C03654=1212.601,101.291,-48.958,-178.587,5.743,148.593
C03655=1212.595,101.540,-48.977,-178.585,5.744,148.593
C03656=1212.591,101.790,-48.996,-178.582,5.744,148.592
C03657=1212.586,102.039,-49.014,-178.579,5.746,148.592
C03658=1212.581,102.288,-49.033,-178.577,5.747,148.591
C03659=1212.577,102.537,-49.052,-178.574,5.747,148.591
C03660=1212.571,102.787,-49.070,-178.572,5.748,148.590
C03661=1212.567,103.035,-49.089,-178.569,5.750,148.590
C03662=1212.561,103.286,-49.108,-178.567,5.750,148.589
C03663=1212.557,103.534,-49.127,-178.564,5.751,148.589
C03664=1212.553,103.784,-49.145,-178.561,5.752,148.588
C03665=1212.547,104.033,-49.164,-178.559,5.753,148.588
C03666=1212.543,104.281,-49.183,-178.556,5.754,148.587
C03667=1212.538,104.532,-49.202,-178.553,5.756,148.587
C03668=1212.533,104.780,-49.221,-178.551,5.756,148.586
C03669=1212.528,105.030,-49.240,-178.549,5.757,148.585
C03670=1212.523,105.279,-49.258,-178.545,5.759,148.585
C03671=1212.519,105.529,-49.278,-178.543,5.760,148.584
C03672=1212.514,105.778,-49.296,-178.541,5.760,148.584
C03673=1212.508,106.027,-49.315,-178.537,5.762,148.583
C03674=1212.504,106.276,-49.334,-178.535,5.763,148.583
C03675=1212.499,106.525,-49.353,-178.533,5.763,148.582
C03676=1212.495,106.775,-49.372,-178.530,5.765,148.582
C03677=1212.489,107.043,-49.393,-178.527,5.766,148.581
C03678=1212.484,107.312,-49.413,-178.524,5.767,148.580
C03679=1212.478,107.580,-49.434,-178.522,5.768,148.580
C03680=1212.474,107.849,-49.454,-178.519,5.769,148.579
C03681=1212.469,108.098,-49.473,-178.516,5.770,148.579
C03682=1212.465,108.347,-49.492,-178.514,5.771,148.578
C03683=1212.459,108.596,-49.511,-178.511,5.772,148.578
C03684=1212.454,108.846,-49.530,-178.509,5.773,148.577
C03685=1212.450,109.094,-49.549,-178.506,5.774,148.577
C03686=1212.444,109.343,-49.568,-178.503,5.775,148.576
C03687=1212.440,109.593,-49.587,-178.501,5.776,148.576
C03688=1212.435,109.842,-49.606,-178.498,5.777,148.575
C03689=1212.430,110.092,-49.625,-178.496,5.779,148.575
C03690=1212.426,110.341,-49.645,-178.493,5.779,148.574
C03691=1212.420,110.590,-49.664,-178.491,5.780,148.573
C03692=1212.416,110.839,-49.683,-178.488,5.782,148.573
C03693=1212.411,111.088,-49.702,-178.486,5.783,148.572
C03694=1212.406,111.338,-49.721,-178.483,5.783,148.572
C03695=1212.401,111.587,-49.740,-178.480,5.785,148.571
C03696=1212.397,111.836,-49.759,-178.478,5.786,148.571
C03697=1212.391,112.085,-49.779,-178.475,5.787,148.570
C03698=1212.387,112.334,-49.798,-178.472,5.788,148.570
C03699=1212.382,112.583,-49.817,-178.470,5.789,148.569
C03700=1212.377,112.833,-49.837,-178.467,5.790,148.569
C03701=1212.373,113.081,-49.855,-178.465,5.791,148.568
C03702=1212.368,113.331,-49.875,-178.462,5.792,148.568
C03703=1212.363,113.581,-49.894,-178.459,5.793,148.567
C03704=1212.358,113.830,-49.913,-178.457,5.794,148.567
C03705=1212.354,114.079,-49.932,-178.454,5.796,148.566
C03706=1212.348,114.328,-49.952,-178.452,5.797,148.566
C03707=1212.343,114.578,-49.971,-178.449,5.797,148.565
C03708=1212.339,114.826,-49.990,-178.446,5.799,148.564
C03709=1212.334,115.076,-50.010,-178.444,5.800,148.564
C03710=1212.329,115.325,-50.029,-178.442,5.801,148.563
C03711=1212.324,115.574,-50.049,-178.439,5.802,148.563
C03712=1212.320,115.823,-50.068,-178.436,5.803,148.562
C03713=1212.315,116.072,-50.087,-178.433,5.804,148.562
C03714=1212.310,116.322,-50.107,-178.431,5.805,148.561
C03715=1212.305,116.571,-50.126,-178.429,5.806,148.561
C03716=1212.300,116.820,-50.146,-178.426,5.808,148.560
C03717=1212.296,117.069,-50.165,-178.423,5.808,148.560
C03718=1212.291,117.319,-50.185,-178.421,5.809,148.559
C03719=1212.286,117.567,-50.204,-178.418,5.811,148.559
C03720=1212.281,117.817,-50.224,-178.416,5.812,148.558
C03721=1212.276,118.066,-50.243,-178.413,5.813,148.558
C03722=1212.272,118.315,-50.262,-178.411,5.814,148.557
C03723=1212.267,118.565,-50.282,-178.408,5.815,148.557
C03724=1212.262,118.814,-50.301,-178.405,5.816,148.556
C03725=1212.257,119.062,-50.322,-178.403,5.817,148.556
C03726=1212.253,119.312,-50.341,-178.400,5.819,148.555
C03727=1212.247,119.561,-50.361,-178.397,5.819,148.554
C03728=1212.243,119.810,-50.380,-178.395,5.820,148.554
C03729=1212.239,120.060,-50.399,-178.392,5.822,148.553
C03730=1212.233,120.309,-50.419,-178.390,5.823,148.553
C03731=1212.229,120.558,-50.439,-178.387,5.824,148.553
C03732=1212.224,120.807,-50.459,-178.385,5.825,148.552
C03733=1212.219,121.056,-50.478,-178.382,5.827,148.552
C03734=1212.214,121.306,-50.498,-178.379,5.827,148.551
C03735=1212.209,121.555,-50.517,-178.377,5.828,148.551
C03736=1212.205,121.804,-50.538,-178.374,5.830,148.550
C03737=1212.199,122.053,-50.557,-178.372,5.831,148.550
C03738=1212.195,122.302,-50.576,-178.369,5.832,148.549
C03739=1212.191,122.551,-50.596,-178.367,5.833,148.549
C03740=1212.186,122.800,-50.616,-178.363,5.835,148.548
C03741=1212.181,123.050,-50.635,-178.361,5.836,148.547
C03742=1212.176,123.299,-50.655,-178.359,5.836,148.547
C03743=1212.172,123.548,-50.675,-178.356,5.838,148.546
C03744=1212.166,123.797,-50.695,-178.353,5.839,148.546
C03745=1212.162,124.047,-50.714,-178.351,5.840,148.545
C03746=1212.157,124.295,-50.735,-178.348,5.841,148.545
C03747=1212.152,124.545,-50.754,-178.345,5.843,148.544
C03748=1212.147,124.793,-50.774,-178.343,5.844,148.544
C03749=1212.143,125.043,-50.794,-178.341,5.844,148.543
C03750=1212.138,125.292,-50.814,-178.338,5.846,148.543
C03751=1212.134,125.541,-50.834,-178.335,5.847,148.542
C03752=1212.128,125.790,-50.853,-178.333,5.849,148.542
C03753=1212.124,126.039,-50.874,-178.330,5.849,148.541
C03754=1212.119,126.289,-50.893,-178.327,5.851,148.541
C03755=1212.114,126.538,-50.913,-178.325,5.852,148.540
C03756=1212.110,126.787,-50.933,-178.322,5.853,148.540
C03757=1212.104,127.036,-50.953,-178.320,5.854,148.539
C03758=1212.100,127.285,-50.973,-178.317,5.855,148.539
C03759=1212.095,127.535,-50.993,-178.315,5.857,148.538
C03760=1212.090,127.784,-51.014,-178.312,5.857,148.538
C03761=1212.085,128.033,-51.033,-178.309,5.859,148.537
C03762=1212.080,128.282,-51.053,-178.307,5.860,148.537
C03763=1212.076,128.531,-51.073,-178.304,5.861,148.536
C03764=1212.071,128.780,-51.093,-178.302,5.862,148.536
C03765=1212.066,129.030,-51.113,-178.299,5.864,148.535
C03766=1212.062,129.279,-51.133,-178.297,5.865,148.535
C03767=1212.057,129.528,-51.153,-178.294,5.866,148.534
C03768=1212.052,129.777,-51.173,-178.291,5.867,148.534
C03769=1212.047,130.026,-51.193,-178.289,5.868,148.533
C03770=1212.042,130.275,-51.214,-178.286,5.870,148.533
C03771=1212.038,130.524,-51.234,-178.284,5.870,148.532
C03772=1212.033,130.774,-51.254,-178.281,5.872,148.532
C03773=1212.029,131.023,-51.274,-178.279,5.873,148.532
C03774=1212.023,131.272,-51.293,-178.276,5.874,148.531
C03775=1212.019,131.521,-51.314,-178.273,5.875,148.530
C03776=1212.014,131.770,-51.335,-178.270,5.877,148.530
C03777=1212.009,132.020,-51.354,-178.268,5.878,148.529
C03778=1212.005,132.268,-51.375,-178.265,5.879,148.529
C03779=1212.000,132.517,-51.395,-178.263,5.880,148.528
C03780=1211.995,132.767,-51.415,-178.260,5.882,148.528
C03781=1211.990,133.035,-51.437,-178.258,5.883,148.527
C03782=1211.984,133.304,-51.459,-178.254,5.884,148.527
C03783=1211.980,133.572,-51.481,-178.252,5.886,148.526
C03784=1211.974,133.841,-51.502,-178.249,5.886,148.526
C03785=1211.970,134.090,-51.523,-178.246,5.888,148.525
C03786=1211.965,134.339,-51.543,-178.244,5.889,148.525
C03787=1211.960,134.588,-51.564,-178.241,5.891,148.524
C03788=1211.955,134.838,-51.584,-178.239,5.892,148.524
C03789=1211.951,135.087,-51.604,-178.236,5.893,148.523
C03790=1211.946,135.336,-51.624,-178.234,5.894,148.523
C03791=1211.941,135.585,-51.645,-178.231,5.895,148.522
C03792=1211.937,135.835,-51.665,-178.229,5.896,148.522
C03793=1211.932,136.084,-51.685,-178.226,5.898,148.522
C03794=1211.927,136.333,-51.706,-178.223,5.900,148.521
C03795=1211.922,136.582,-51.727,-178.221,5.901,148.521
C03796=1211.917,136.830,-51.747,-178.217,5.902,148.520
C03797=1211.912,137.079,-51.768,-178.215,5.903,148.520
C03798=1211.907,137.329,-51.787,-178.213,5.905,148.519
C03799=1211.903,137.578,-51.808,-178.210,5.905,148.519
C03800=1211.898,137.827,-51.829,-178.207,5.907,148.518
C03801=1211.893,138.076,-51.849,-178.205,5.908,148.518
C03802=1211.889,138.325,-51.869,-178.202,5.910,148.517
C03803=1211.884,138.574,-51.890,-178.200,5.911,148.517
C03804=1211.879,138.823,-51.911,-178.197,5.912,148.516
C03805=1211.875,139.072,-51.931,-178.195,5.913,148.516
C03806=1211.870,139.321,-51.952,-178.192,5.915,148.515
C03807=1211.865,139.570,-51.972,-178.189,5.915,148.515
C03808=1211.860,139.820,-51.993,-178.187,5.917,148.514
C03809=1211.855,140.069,-52.013,-178.185,5.918,148.514
C03810=1211.851,140.318,-52.033,-178.181,5.920,148.513
C03811=1211.846,140.567,-52.054,-178.179,5.921,148.513
C03812=1211.841,140.816,-52.075,-178.176,5.922,148.512
C03813=1211.836,141.066,-52.096,-178.174,5.923,148.512
C03814=1211.832,141.315,-52.116,-178.171,5.925,148.512
C03815=1211.827,141.564,-52.137,-178.168,5.926,148.511
C03816=1211.823,141.814,-52.158,-178.166,5.927,148.511
C03817=1211.819,142.062,-52.179,-178.163,5.929,148.510
C03818=1211.813,142.311,-52.200,-178.161,5.930,148.510
C03819=1211.809,142.560,-52.220,-178.158,5.931,148.509
C03820=1211.804,142.809,-52.241,-178.156,5.932,148.509
C03821=1211.799,143.058,-52.262,-178.153,5.934,148.508
C03822=1211.794,143.308,-52.283,-178.151,5.935,148.508
C03823=1211.790,143.556,-52.303,-178.148,5.937,148.507
C03824=1211.785,143.806,-52.324,-178.145,5.937,148.507
C03825=1211.780,144.055,-52.344,-178.143,5.939,148.506
C03826=1211.775,144.304,-52.365,-178.140,5.941,148.506
C03827=1211.771,144.552,-52.386,-178.138,5.942,148.505
C03828=1211.766,144.802,-52.407,-178.135,5.943,148.505
C03829=1211.762,145.051,-52.428,-178.132,5.944,148.504
C03830=1211.757,145.300,-52.449,-178.130,5.946,148.504
C03831=1211.752,145.549,-52.469,-178.127,5.947,148.504
C03832=1211.747,145.799,-52.490,-178.124,5.948,148.503
C03833=1211.742,146.047,-52.512,-178.122,5.950,148.503
C03834=1211.738,146.296,-52.532,-178.120,5.951,148.502
C03835=1211.733,146.546,-52.553,-178.116,5.952,148.502
C03836=1211.728,146.794,-52.574,-178.114,5.953,148.501
C03837=1211.723,147.044,-52.595,-178.112,5.955,148.501
C03838=1211.719,147.293,-52.617,-178.109,5.956,148.500
C03839=1211.714,147.542,-52.637,-178.106,5.958,148.500
C03840=1211.709,147.791,-52.658,-178.104,5.959,148.499
C03841=1211.705,148.040,-52.679,-178.101,5.960,148.499
C03842=1211.700,148.289,-52.700,-178.098,5.962,148.498
C03843=1211.695,148.538,-52.721,-178.096,5.963,148.498
C03844=1211.691,148.788,-52.742,-178.094,5.965,148.498
C03845=1211.686,149.036,-52.764,-178.091,5.965,148.497
C03846=1211.681,149.286,-52.784,-178.088,5.967,148.497
C03847=1211.676,149.535,-52.805,-178.086,5.969,148.496
C03848=1211.671,149.783,-52.827,-178.083,5.969,148.496
C03849=1211.666,150.033,-52.848,-178.080,5.971,148.495
C03850=1211.663,150.282,-52.869,-178.078,5.972,148.495
C03851=1211.658,150.531,-52.890,-178.075,5.974,148.494
C03852=1211.652,150.780,-52.911,-178.072,5.975,148.494
C03853=1211.648,151.028,-52.932,-178.070,5.976,148.494
C03854=1211.643,151.278,-52.953,-178.067,5.978,148.493
C03855=1211.639,151.527,-52.975,-178.065,5.979,148.493
C03856=1211.634,151.776,-52.995,-178.062,5.981,148.492
C03857=1211.629,152.025,-53.016,-178.060,5.982,148.492
C03858=1211.624,152.274,-53.038,-178.057,5.983,148.491
C03859=1211.619,152.523,-53.059,-178.054,5.985,148.491
C03860=1211.616,152.772,-53.080,-178.052,5.986,148.490
C03861=1211.610,153.021,-53.101,-178.049,5.987,148.490
C03862=1211.606,153.270,-53.123,-178.047,5.989,148.489
C03863=1211.600,153.519,-53.144,-178.044,5.990,148.489
C03864=1211.596,153.769,-53.166,-178.041,5.992,148.488
C03865=1211.592,154.018,-53.186,-178.039,5.993,148.488
C03866=1211.587,154.266,-53.208,-178.036,5.994,148.488
C03867=1211.582,154.515,-53.229,-178.034,5.996,148.487
C03868=1211.577,154.765,-53.251,-178.031,5.997,148.487
C03869=1211.573,155.013,-53.273,-178.029,5.999,148.486
C03870=1211.568,155.262,-53.293,-178.026,6.000,148.486
C03871=1211.564,155.512,-53.315,-178.023,6.001,148.485
C03872=1211.559,155.761,-53.336,-178.021,6.003,148.485
C03873=1211.554,156.010,-53.358,-178.018,6.005,148.485
C03874=1211.549,156.259,-53.379,-178.016,6.006,148.484
C03875=1211.544,156.508,-53.401,-178.013,6.007,148.484
C03876=1211.540,156.757,-53.422,-178.011,6.008,148.483
C03877=1211.535,157.006,-53.443,-178.008,6.010,148.483
C03878=1211.531,157.255,-53.465,-178.005,6.012,148.482
C03879=1211.526,157.504,-53.487,-178.003,6.012,148.482
C03880=1211.521,157.753,-53.508,-178.000,6.014,148.481
C03881=1211.516,158.002,-53.530,-177.997,6.016,148.481
C03882=1211.512,158.251,-53.551,-177.995,6.017,148.481
C03883=1211.506,158.500,-53.572,-177.992,6.018,148.480
C03884=1211.502,158.750,-53.594,-177.989,6.020,148.480
C03885=1211.497,159.019,-53.617,-177.987,6.022,148.479
C03886=1211.492,159.287,-53.641,-177.984,6.023,148.479
C03887=1211.487,159.557,-53.664,-177.981,6.024,148.478
C03888=1211.482,159.826,-53.687,-177.978,6.026,148.478
C03889=1211.477,160.075,-53.709,-177.976,6.028,148.477
C03890=1211.472,160.323,-53.731,-177.974,6.029,148.477
C03891=1211.468,160.573,-53.753,-177.971,6.030,148.477
C03892=1211.463,160.821,-53.774,-177.968,6.032,148.476
C03893=1211.458,161.070,-53.795,-177.966,6.033,148.476
C03894=1211.454,161.320,-53.818,-177.963,6.035,148.475
C03895=1211.449,161.568,-53.839,-177.960,6.036,148.475
C03896=1211.445,161.818,-53.861,-177.958,6.037,148.474
C03897=1211.440,162.066,-53.883,-177.955,6.039,148.474
C03898=1211.435,162.315,-53.905,-177.952,6.041,148.474
C03899=1211.430,162.565,-53.926,-177.950,6.042,148.473
C03900=1211.425,162.814,-53.948,-177.947,6.043,148.473
C03901=1211.421,163.063,-53.970,-177.944,6.045,148.472
C03902=1211.416,163.312,-53.991,-177.942,6.046,148.472
C03903=1211.411,163.560,-54.013,-177.940,6.048,148.471
C03904=1211.407,163.810,-54.035,-177.937,6.049,148.471
C03905=1211.402,164.058,-54.057,-177.934,6.051,148.471
C03906=1211.398,164.308,-54.079,-177.932,6.052,148.470
C03907=1211.393,164.556,-54.100,-177.929,6.054,148.470
C03908=1211.389,164.806,-54.123,-177.926,6.056,148.469
C03909=1211.384,165.054,-54.144,-177.924,6.056,148.469
C03910=1211.379,165.303,-54.166,-177.921,6.058,148.468
C03911=1211.375,165.552,-54.188,-177.919,6.060,148.468
C03912=1211.370,165.801,-54.210,-177.916,6.061,148.468
C03913=1211.365,166.050,-54.232,-177.914,6.063,148.467
C03914=1211.360,166.299,-54.254,-177.911,6.064,148.467
C03915=1211.356,166.548,-54.276,-177.908,6.065,148.466
C03916=1211.351,166.797,-54.298,-177.906,6.067,148.466
C03917=1211.347,167.046,-54.320,-177.903,6.069,148.466
C03918=1211.342,167.295,-54.341,-177.900,6.070,148.465
C03919=1211.337,167.544,-54.363,-177.898,6.071,148.465
C03920=1211.332,167.793,-54.386,-177.895,6.073,148.464
C03921=1211.328,168.043,-54.408,-177.893,6.075,148.464
C03922=1211.323,168.291,-54.429,-177.890,6.076,148.463
C03923=1211.318,168.541,-54.452,-177.887,6.077,148.463
C03924=1211.314,168.789,-54.474,-177.885,6.079,148.463
C03925=1211.309,169.038,-54.497,-177.882,6.081,148.462
C03926=1211.304,169.287,-54.518,-177.880,6.082,148.462
C03927=1211.300,169.536,-54.540,-177.877,6.084,148.461
C03928=1211.295,169.785,-54.562,-177.875,6.086,148.461
C03929=1211.291,170.034,-54.584,-177.872,6.086,148.460
C03930=1211.285,170.283,-54.607,-177.869,6.088,148.460
C03931=1211.281,170.532,-54.629,-177.867,6.090,148.460
C03932=1211.277,170.781,-54.651,-177.864,6.092,148.459
C03933=1211.272,171.030,-54.673,-177.862,6.093,148.459
C03934=1211.267,171.280,-54.695,-177.859,6.094,148.458
C03935=1211.262,171.528,-54.718,-177.856,6.096,148.458
C03936=1211.258,171.777,-54.740,-177.853,6.098,148.458
C03937=1211.252,172.026,-54.762,-177.851,6.099,148.457
C03938=1211.248,172.275,-54.784,-177.849,6.101,148.457
C03939=1211.244,172.523,-54.807,-177.846,6.102,148.457
C03940=1211.239,172.773,-54.829,-177.843,6.103,148.456
C03941=1211.234,173.022,-54.851,-177.841,6.105,148.456
C03942=1211.230,173.270,-54.874,-177.838,6.107,148.455
C03943=1211.226,173.520,-54.896,-177.835,6.108,148.455
C03944=1211.220,173.769,-54.918,-177.833,6.109,148.454
C03945=1211.216,174.017,-54.941,-177.831,6.111,148.454
C03946=1211.212,174.267,-54.963,-177.828,6.113,148.454
C03947=1211.206,174.516,-54.985,-177.825,6.115,148.453
C03948=1211.202,174.764,-55.008,-177.823,6.115,148.453
C03949=1211.197,175.013,-55.030,-177.820,6.117,148.452
C03950=1211.193,175.262,-55.053,-177.817,6.119,148.452
C03951=1211.188,175.511,-55.075,-177.815,6.121,148.452
C03952=1211.183,175.760,-55.097,-177.812,6.122,148.451
C03953=1211.179,176.009,-55.120,-177.810,6.123,148.451
C03954=1211.174,176.259,-55.143,-177.807,6.125,148.450
C03955=1211.169,176.507,-55.165,-177.804,6.127,148.450
C03956=1211.165,176.756,-55.187,-177.802,6.129,148.450
C03957=1211.160,177.005,-55.210,-177.799,6.130,148.449
C03958=1211.155,177.254,-55.232,-177.797,6.132,148.449
C03959=1211.151,177.503,-55.256,-177.794,6.133,148.448
C03960=1211.146,177.752,-55.278,-177.791,6.135,148.448
C03961=1211.141,178.000,-55.301,-177.789,6.136,148.448
C03962=1211.137,178.250,-55.323,-177.786,6.138,148.447
C03963=1211.133,178.498,-55.345,-177.784,6.140,148.447
C03964=1211.127,178.747,-55.368,-177.781,6.141,148.447
C03965=1211.123,178.996,-55.390,-177.778,6.143,148.446
C03966=1211.118,179.246,-55.413,-177.776,6.144,148.446
C03967=1211.114,179.494,-55.435,-177.773,6.146,148.445
C03968=1211.109,179.743,-55.458,-177.770,6.148,148.445
C03969=1211.105,179.992,-55.481,-177.768,6.149,148.444
C03970=1211.100,180.241,-55.504,-177.766,6.150,148.444
C03971=1211.095,180.490,-55.526,-177.763,6.152,148.444
C03972=1211.090,180.739,-55.549,-177.760,6.154,148.443
C03973=1211.086,180.988,-55.573,-177.758,6.156,148.443
C03974=1211.081,181.237,-55.594,-177.755,6.158,148.443
C03975=1211.076,181.486,-55.618,-177.752,6.158,148.442
C03976=1211.072,181.734,-55.640,-177.750,6.160,148.442
C03977=1211.067,181.984,-55.663,-177.747,6.162,148.441
C03978=1211.063,182.232,-55.685,-177.744,6.164,148.441
C03979=1211.058,182.481,-55.709,-177.742,6.166,148.441
C03980=1211.054,182.730,-55.731,-177.740,6.167,148.440
C03981=1211.049,182.979,-55.754,-177.737,6.168,148.440
C03982=1211.044,183.228,-55.778,-177.734,6.170,148.440
C03983=1211.040,183.476,-55.800,-177.732,6.172,148.439
C03984=1211.035,183.726,-55.823,-177.729,6.174,148.439
C03985=1211.031,183.975,-55.845,-177.727,6.174,148.438
C03986=1211.026,184.224,-55.869,-177.724,6.176,148.438
C03987=1211.021,184.472,-55.892,-177.721,6.178,148.438
C03988=1211.016,184.722,-55.914,-177.719,6.180,148.437
C03989=1211.011,184.991,-55.940,-177.716,6.182,148.437
C03990=1211.006,185.260,-55.965,-177.713,6.184,148.436
C03991=1211.002,185.530,-55.989,-177.710,6.185,148.436
C03992=1210.996,185.800,-56.014,-177.707,6.187,148.436
C03993=1210.992,186.049,-56.037,-177.705,6.189,148.435
C03994=1210.987,186.298,-56.059,-177.702,6.191,148.435
C03995=1210.983,186.547,-56.083,-177.700,6.192,148.434
C03996=1210.978,186.796,-56.106,-177.697,6.194,148.434
C03997=1210.973,187.044,-56.129,-177.695,6.195,148.434
C03998=1210.969,187.293,-56.152,-177.692,6.197,148.433
C03999=1210.964,187.542,-56.175,-177.689,6.199,148.433
C04000=1210.959,187.791,-56.199,-177.686,6.200,148.432
C04001=1210.955,188.040,-56.221,-177.684,6.202,148.432
C04002=1210.951,188.289,-56.245,-177.681,6.204,148.432
C04003=1210.946,188.538,-56.268,-177.679,6.205,148.431
C04004=1210.941,188.786,-56.291,-177.676,6.207,148.431
C04005=1210.937,189.035,-56.314,-177.674,6.209,148.431
C04006=1210.932,189.284,-56.337,-177.671,6.210,148.430
C04007=1210.927,189.533,-56.361,-177.668,6.212,148.430
C04008=1210.923,189.782,-56.384,-177.666,6.214,148.430
C04009=1210.919,190.031,-56.407,-177.664,6.215,148.429
C04010=1210.914,190.280,-56.430,-177.661,6.217,148.429
C04011=1210.909,190.529,-56.453,-177.658,6.219,148.429
C04012=1210.904,190.778,-56.477,-177.656,6.221,148.428
C04013=1210.899,191.026,-56.500,-177.653,6.222,148.428
C04014=1210.894,191.275,-56.523,-177.650,6.224,148.428
C04015=1210.890,191.524,-56.546,-177.648,6.226,148.427
C04016=1210.886,191.773,-56.569,-177.645,6.228,148.427
C04017=1210.881,192.022,-56.593,-177.643,6.229,148.426
C04018=1210.876,192.271,-56.616,-177.640,6.230,148.426
C04019=1210.872,192.520,-56.640,-177.637,6.232,148.426
C04020=1210.867,192.769,-56.663,-177.634,6.234,148.425
C04021=1210.863,193.018,-56.687,-177.632,6.236,148.425
C04022=1210.858,193.267,-56.710,-177.629,6.238,148.424
C04023=1210.854,193.515,-56.733,-177.627,6.239,148.424
C04024=1210.849,193.764,-56.756,-177.624,6.241,148.424
C04025=1210.845,194.013,-56.780,-177.622,6.242,148.423
C04026=1210.840,194.262,-56.804,-177.619,6.244,148.423
C04027=1210.835,194.511,-56.827,-177.616,6.246,148.423
C04028=1210.831,194.760,-56.850,-177.614,6.248,148.422
C04029=1210.826,195.009,-56.874,-177.611,6.250,148.422
C04030=1210.822,195.257,-56.898,-177.609,6.251,148.422
C04031=1210.817,195.506,-56.921,-177.606,6.253,148.421
C04032=1210.812,195.755,-56.945,-177.603,6.255,148.421
C04033=1210.808,196.004,-56.969,-177.601,6.256,148.421
C04034=1210.803,196.253,-56.992,-177.598,6.258,148.420
C04035=1210.798,196.502,-57.015,-177.596,6.260,148.420
C04036=1210.794,196.751,-57.039,-177.593,6.262,148.420
C04037=1210.789,196.999,-57.063,-177.591,6.263,148.419
C04038=1210.785,197.248,-57.086,-177.588,6.265,148.419
C04039=1210.780,197.497,-57.110,-177.585,6.267,148.419
C04040=1210.776,197.746,-57.134,-177.583,6.269,148.418
C04041=1210.771,197.995,-57.157,-177.580,6.271,148.418
C04042=1210.766,198.243,-57.181,-177.577,6.272,148.418
C04043=1210.762,198.492,-57.204,-177.575,6.274,148.417
C04044=1210.757,198.741,-57.228,-177.573,6.275,148.417
C04045=1210.753,198.990,-57.252,-177.570,6.277,148.416
C04046=1210.748,199.239,-57.275,-177.567,6.279,148.416
C04047=1210.744,199.487,-57.299,-177.565,6.281,148.416
C04048=1210.739,199.736,-57.323,-177.562,6.283,148.415
C04049=1210.734,199.985,-57.346,-177.559,6.284,148.415
C04050=1210.730,200.234,-57.370,-177.557,6.286,148.415
C04051=1210.724,200.483,-57.394,-177.554,6.288,148.414
C04052=1210.720,200.731,-57.418,-177.551,6.290,148.414
C04053=1210.715,200.980,-57.441,-177.549,6.292,148.414
C04054=1210.711,201.230,-57.466,-177.546,6.294,148.413
C04055=1210.707,201.479,-57.489,-177.543,6.295,148.413
C04056=1210.702,201.727,-57.513,-177.541,6.297,148.413
C04057=1210.698,201.975,-57.537,-177.539,6.298,148.412
C04058=1210.693,202.224,-57.561,-177.536,6.300,148.412
C04059=1210.688,202.473,-57.585,-177.533,6.302,148.412
C04060=1210.683,202.722,-57.609,-177.531,6.304,148.411
C04061=1210.679,202.971,-57.633,-177.528,6.306,148.411
C04062=1210.674,203.220,-57.656,-177.525,6.307,148.411
C04063=1210.671,203.469,-57.681,-177.523,6.309,148.410
C04064=1210.665,203.717,-57.705,-177.520,6.311,148.410
C04065=1210.661,203.967,-57.729,-177.518,6.313,148.410
C04066=1210.656,204.215,-57.753,-177.515,6.315,148.409
C04067=1210.652,204.463,-57.777,-177.512,6.317,148.409
C04068=1210.647,204.712,-57.800,-177.510,6.318,148.409
C04069=1210.643,204.962,-57.825,-177.507,6.320,148.408
C04070=1210.638,205.210,-57.849,-177.504,6.322,148.408
C04071=1210.634,205.459,-57.873,-177.502,6.324,148.408
C04072=1210.629,205.708,-57.897,-177.500,6.326,148.407
C04073=1210.624,205.956,-57.921,-177.497,6.328,148.407
C04074=1210.619,206.205,-57.945,-177.494,6.330,148.407
C04075=1210.616,206.455,-57.969,-177.492,6.332,148.406
C04076=1210.611,206.703,-57.993,-177.489,6.333,148.406
C04077=1210.606,206.952,-58.018,-177.487,6.334,148.406
C04078=1210.601,207.201,-58.041,-177.484,6.336,148.405
C04079=1210.597,207.449,-58.065,-177.482,6.338,148.405
C04080=1210.592,207.699,-58.090,-177.479,6.340,148.405
C04081=1210.588,207.947,-58.114,-177.476,6.342,148.404
C04082=1210.584,208.195,-58.139,-177.474,6.344,148.404
C04083=1210.578,208.445,-58.162,-177.471,6.345,148.404
C04084=1210.574,208.693,-58.187,-177.468,6.347,148.403
C04085=1210.570,208.942,-58.211,-177.466,6.349,148.403
C04086=1210.565,209.191,-58.236,-177.463,6.351,148.403
C04087=1210.561,209.439,-58.260,-177.460,6.353,148.402
C04088=1210.556,209.688,-58.284,-177.458,6.355,148.402
C04089=1210.552,209.937,-58.309,-177.456,6.357,148.402
C04090=1210.547,210.186,-58.333,-177.453,6.359,148.402
C04091=1210.542,210.435,-58.357,-177.450,6.360,148.401
C04092=1210.537,210.683,-58.381,-177.448,6.362,148.401
C04093=1210.533,210.954,-58.408,-177.445,6.364,148.401
C04094=1210.528,211.224,-58.435,-177.442,6.367,148.400
C04095=1210.523,211.494,-58.461,-177.439,6.369,148.400
C04096=1210.518,211.765,-58.487,-177.436,6.370,148.399
C04097=1210.513,212.014,-58.512,-177.434,6.372,148.399
C04098=1210.509,212.263,-58.536,-177.431,6.374,148.399
C04099=1210.504,212.512,-58.561,-177.429,6.376,148.399
C04100=1210.499,212.760,-58.585,-177.426,6.378,148.398
C04101=1210.495,213.009,-58.610,-177.423,6.380,148.398
C04102=1210.491,213.257,-58.635,-177.421,6.382,148.398
C04103=1210.486,213.506,-58.659,-177.418,6.383,148.397
C04104=1210.482,213.755,-58.684,-177.415,6.385,148.397
C04105=1210.477,214.004,-58.708,-177.413,6.387,148.397
C04106=1210.472,214.252,-58.732,-177.410,6.389,148.396
C04107=1210.468,214.502,-58.757,-177.408,6.391,148.396
C04108=1210.463,214.750,-58.782,-177.405,6.393,148.396
C04109=1210.458,214.999,-58.806,-177.403,6.395,148.395
C04110=1210.454,215.248,-58.831,-177.400,6.397,148.395
C04111=1210.449,215.497,-58.855,-177.397,6.398,148.395
C04112=1210.445,215.744,-58.880,-177.395,6.400,148.394
C04113=1210.441,215.994,-58.905,-177.392,6.403,148.394
C04114=1210.436,216.242,-58.929,-177.389,6.405,148.394
C04115=1210.432,216.492,-58.954,-177.386,6.407,148.393
C04116=1210.427,216.740,-58.979,-177.384,6.409,148.393
C04117=1210.422,216.989,-59.003,-177.382,6.411,148.393
C04118=1210.418,217.238,-59.029,-177.379,6.412,148.393
C04119=1210.414,217.486,-59.053,-177.376,6.414,148.392
C04120=1210.409,217.735,-59.078,-177.374,6.416,148.392
C04121=1210.404,217.984,-59.102,-177.371,6.418,148.392
C04122=1210.400,218.232,-59.127,-177.368,6.420,148.391
C04123=1210.395,218.481,-59.152,-177.366,6.422,148.391
C04124=1210.391,218.730,-59.176,-177.364,6.424,148.391
C04125=1210.387,218.979,-59.202,-177.361,6.426,148.391
C04126=1210.382,219.227,-59.227,-177.358,6.428,148.390
C04127=1210.377,219.476,-59.251,-177.356,6.429,148.390
C04128=1210.373,219.725,-59.276,-177.353,6.431,148.390
C04129=1210.368,219.973,-59.301,-177.350,6.433,148.389
C04130=1210.364,220.222,-59.326,-177.348,6.435,148.389
C04131=1210.359,220.470,-59.351,-177.346,6.437,148.389
C04132=1210.355,220.720,-59.376,-177.343,6.439,148.389
C04133=1210.350,220.968,-59.400,-177.340,6.441,148.388
C04134=1210.346,221.217,-59.426,-177.338,6.443,148.388
C04135=1210.341,221.466,-59.451,-177.335,6.444,148.388
C04136=1210.337,221.715,-59.476,-177.332,6.446,148.387
C04137=1210.332,221.963,-59.500,-177.330,6.449,148.387
C04138=1210.327,222.212,-59.525,-177.327,6.451,148.387
C04139=1210.323,222.461,-59.551,-177.324,6.453,148.386
C04140=1210.318,222.709,-59.576,-177.322,6.455,148.386
C04141=1210.314,222.958,-59.601,-177.319,6.457,148.386
C04142=1210.309,223.207,-59.625,-177.317,6.458,148.385
C04143=1210.305,223.455,-59.651,-177.314,6.461,148.385
C04144=1210.300,223.704,-59.676,-177.312,6.463,148.385
C04145=1210.296,223.953,-59.702,-177.309,6.464,148.385
C04146=1210.291,224.201,-59.726,-177.306,6.466,148.384
C04147=1210.287,224.450,-59.751,-177.304,6.468,148.384
C04148=1210.282,224.699,-59.776,-177.301,6.470,148.384
C04149=1210.278,224.948,-59.802,-177.299,6.472,148.384
C04150=1210.273,225.196,-59.828,-177.296,6.474,148.383
C04151=1210.269,225.445,-59.852,-177.294,6.476,148.383
C04152=1210.265,225.694,-59.877,-177.291,6.478,148.383
C04153=1210.260,225.942,-59.902,-177.288,6.480,148.382
C04154=1210.255,226.191,-59.928,-177.286,6.482,148.382
C04155=1210.251,226.439,-59.953,-177.283,6.484,148.382
C04156=1210.246,226.689,-59.978,-177.281,6.486,148.382
C04157=1210.241,226.937,-60.004,-177.278,6.488,148.381
C04158=1210.237,227.186,-60.029,-177.275,6.490,148.381
C04159=1210.233,227.435,-60.054,-177.273,6.492,148.381
C04160=1210.228,227.683,-60.079,-177.270,6.494,148.381
C04161=1210.224,227.932,-60.105,-177.268,6.496,148.380
C04162=1210.219,228.180,-60.130,-177.265,6.498,148.380
C04163=1210.215,228.429,-60.155,-177.263,6.500,148.380
C04164=1210.210,228.677,-60.181,-177.260,6.502,148.379
C04165=1210.205,228.927,-60.206,-177.258,6.503,148.379
C04166=1210.201,229.175,-60.232,-177.255,6.506,148.379
C04167=1210.196,229.424,-60.257,-177.252,6.508,148.379
C04168=1210.192,229.672,-60.283,-177.250,6.510,148.378
C04169=1210.188,229.921,-60.308,-177.247,6.512,148.378
C04170=1210.183,230.170,-60.333,-177.245,6.514,148.378
C04171=1210.179,230.419,-60.359,-177.242,6.516,148.377
C04172=1210.174,230.667,-60.384,-177.240,6.518,148.377
C04173=1210.170,230.916,-60.410,-177.237,6.520,148.377
C04174=1210.165,231.164,-60.436,-177.235,6.522,148.377
C04175=1210.161,231.413,-60.461,-177.232,6.523,148.376
C04176=1210.156,231.662,-60.486,-177.229,6.526,148.376
C04177=1210.152,231.911,-60.512,-177.227,6.528,148.376
C04178=1210.147,232.159,-60.537,-177.224,6.530,148.376
C04179=1210.143,232.408,-60.563,-177.221,6.532,148.375
C04180=1210.138,232.656,-60.589,-177.219,6.534,148.375
C04181=1210.134,232.905,-60.614,-177.216,6.536,148.375
C04182=1210.129,233.153,-60.640,-177.214,6.538,148.375
C04183=1210.125,233.402,-60.666,-177.211,6.540,148.374
C04184=1210.120,233.650,-60.691,-177.209,6.542,148.374
C04185=1210.115,233.899,-60.717,-177.206,6.545,148.374
C04186=1210.111,234.148,-60.743,-177.203,6.546,148.374
C04187=1210.106,234.396,-60.769,-177.201,6.548,148.373
C04188=1210.102,234.645,-60.794,-177.198,6.550,148.373
C04189=1210.098,234.894,-60.820,-177.196,6.552,148.373
C04190=1210.094,235.143,-60.846,-177.193,6.554,148.372
C04191=1210.089,235.391,-60.871,-177.191,6.556,148.372
C04192=1210.085,235.640,-60.897,-177.188,6.558,148.372
C04193=1210.080,235.889,-60.923,-177.186,6.560,148.372
C04194=1210.075,236.138,-60.949,-177.183,6.563,148.371
C04195=1210.071,236.386,-60.974,-177.180,6.565,148.371
C04196=1210.066,236.634,-61.000,-177.178,6.567,148.371
C04197=1210.062,236.906,-61.028,-177.175,6.569,148.371
C04198=1210.057,237.177,-61.057,-177.172,6.571,148.370
C04199=1210.052,237.449,-61.085,-177.169,6.573,148.370
C04200=1210.046,237.720,-61.114,-177.167,6.576,148.370
C04201=1210.042,237.969,-61.139,-177.164,6.578,148.370
C04202=1210.038,238.217,-61.165,-177.161,6.580,148.369
C04203=1210.034,238.466,-61.191,-177.159,6.582,148.369
C04204=1210.029,238.715,-61.217,-177.157,6.584,148.369
C04205=1210.024,238.963,-61.243,-177.154,6.586,148.369
C04206=1210.020,239.212,-61.269,-177.151,6.588,148.368
C04207=1210.016,239.460,-61.295,-177.149,6.591,148.368
C04208=1210.011,239.709,-61.321,-177.146,6.592,148.368
C04209=1210.007,239.958,-61.347,-177.143,6.594,148.368
C04210=1210.002,240.206,-61.373,-177.141,6.596,148.368
C04211=1209.998,240.455,-61.399,-177.139,6.598,148.367
C04212=1209.993,240.704,-61.425,-177.136,6.600,148.367
C04213=1209.989,240.952,-61.451,-177.134,6.602,148.367
C04214=1209.985,241.201,-61.477,-177.131,6.605,148.367
C04215=1209.979,241.449,-61.503,-177.128,6.607,148.366
C04216=1209.975,241.698,-61.529,-177.126,6.609,148.366
C04217=1209.971,241.946,-61.556,-177.123,6.611,148.366
C04218=1209.966,242.195,-61.582,-177.121,6.613,148.366
C04219=1209.962,242.444,-61.608,-177.119,6.615,148.365
C04220=1209.958,242.692,-61.634,-177.115,6.618,148.365
C04221=1209.953,242.941,-61.660,-177.113,6.619,148.365
C04222=1209.948,243.189,-61.687,-177.111,6.622,148.365
C04223=1209.944,243.438,-61.712,-177.108,6.623,148.364
C04224=1209.939,243.687,-61.739,-177.105,6.625,148.364
C04225=1209.935,243.935,-61.765,-177.103,6.628,148.364
C04226=1209.930,244.184,-61.791,-177.100,6.630,148.364
C04227=1209.926,244.432,-61.818,-177.097,6.632,148.363
C04228=1209.922,244.681,-61.844,-177.095,6.634,148.363
C04229=1209.917,244.929,-61.871,-177.093,6.636,148.363
C04230=1209.913,245.178,-61.896,-177.090,6.638,148.363
C04231=1209.908,245.426,-61.923,-177.087,6.641,148.363
C04232=1209.904,245.675,-61.949,-177.085,6.643,148.362
C04233=1209.899,245.923,-61.976,-177.083,6.645,148.362
C04234=1209.895,246.172,-62.002,-177.080,6.647,148.362
C04235=1209.890,246.421,-62.029,-177.077,6.649,148.362
C04236=1209.886,246.669,-62.055,-177.075,6.651,148.362
C04237=1209.881,246.918,-62.082,-177.072,6.654,148.361
C04238=1209.877,247.167,-62.107,-177.069,6.655,148.361
C04239=1209.872,247.415,-62.134,-177.067,6.658,148.361
C04240=1209.869,247.663,-62.161,-177.065,6.659,148.361
C04241=1209.864,247.913,-62.187,-177.062,6.662,148.360
C04242=1209.860,248.161,-62.214,-177.059,6.664,148.360
C04243=1209.855,248.410,-62.240,-177.057,6.666,148.360
C04244=1209.851,248.658,-62.267,-177.054,6.668,148.360
C04245=1209.846,248.907,-62.294,-177.052,6.670,148.359
C04246=1209.842,249.155,-62.319,-177.049,6.673,148.359
C04247=1209.837,249.404,-62.346,-177.047,6.675,148.359
C04248=1209.833,249.652,-62.373,-177.044,6.677,148.359
C04249=1209.828,249.901,-62.399,-177.042,6.679,148.359
C04250=1209.824,250.150,-62.426,-177.039,6.681,148.358
C04251=1209.820,250.398,-62.453,-177.036,6.684,148.358
C04252=1209.815,250.646,-62.480,-177.034,6.686,148.358
C04253=1209.811,250.895,-62.506,-177.031,6.688,148.358
C04254=1209.806,251.144,-62.533,-177.029,6.690,148.358
C04255=1209.802,251.392,-62.560,-177.026,6.692,148.357
C04256=1209.798,251.640,-62.586,-177.024,6.695,148.357
C04257=1209.793,251.889,-62.612,-177.021,6.697,148.357
C04258=1209.788,252.138,-62.640,-177.018,6.699,148.357
C04259=1209.784,252.386,-62.666,-177.016,6.701,148.357
C04260=1209.779,252.635,-62.693,-177.013,6.703,148.356
C04261=1209.775,252.883,-62.720,-177.011,6.706,148.356
C04262=1209.771,253.131,-62.747,-177.008,6.707,148.356
C04263=1209.766,253.380,-62.773,-177.006,6.710,148.356
C04264=1209.761,253.629,-62.800,-177.003,6.712,148.356
C04265=1209.757,253.877,-62.826,-177.001,6.714,148.355
C04266=1209.753,254.126,-62.854,-176.998,6.716,148.355
C04267=1209.748,254.374,-62.881,-176.996,6.718,148.355
C04268=1209.743,254.623,-62.908,-176.993,6.721,148.355
C04269=1209.739,254.871,-62.934,-176.990,6.723,148.355
C04270=1209.735,255.119,-62.961,-176.988,6.725,148.354
C04271=1209.730,255.368,-62.988,-176.986,6.727,148.354
C04272=1209.727,255.617,-63.015,-176.983,6.730,148.354
C04273=1209.722,255.865,-63.042,-176.980,6.732,148.354
C04274=1209.718,256.114,-63.069,-176.978,6.734,148.354
C04275=1209.713,256.362,-63.096,-176.976,6.736,148.353
C04276=1209.708,256.611,-63.123,-176.972,6.739,148.353
C04277=1209.704,256.859,-63.150,-176.970,6.741,148.353
C04278=1209.700,257.107,-63.177,-176.968,6.743,148.353
C04279=1209.695,257.356,-63.204,-176.965,6.745,148.353
C04280=1209.691,257.605,-63.231,-176.962,6.748,148.352
C04281=1209.686,257.853,-63.258,-176.960,6.750,148.352
C04282=1209.682,258.102,-63.285,-176.958,6.752,148.352
C04283=1209.678,258.350,-63.312,-176.955,6.754,148.352
C04284=1209.673,258.599,-63.339,-176.952,6.757,148.352
C04285=1209.668,258.847,-63.366,-176.950,6.759,148.352
C04286=1209.664,259.095,-63.394,-176.947,6.761,148.351
C04287=1209.660,259.344,-63.421,-176.945,6.764,148.351
C04288=1209.655,259.593,-63.448,-176.942,6.766,148.351
C04289=1209.651,259.841,-63.475,-176.940,6.768,148.351
C04290=1209.647,260.089,-63.502,-176.937,6.770,148.350
C04291=1209.642,260.338,-63.529,-176.935,6.773,148.350
C04292=1209.638,260.586,-63.557,-176.932,6.774,148.350
C04293=1209.634,260.835,-63.584,-176.930,6.777,148.350
C04294=1209.629,261.083,-63.611,-176.927,6.779,148.350
C04295=1209.624,261.332,-63.638,-176.925,6.782,148.350
C04296=1209.620,261.580,-63.665,-176.922,6.783,148.349
C04297=1209.615,261.828,-63.693,-176.920,6.786,148.349
C04298=1209.611,262.078,-63.720,-176.917,6.788,148.349
C04299=1209.607,262.326,-63.748,-176.915,6.790,148.349
C04300=1209.602,262.574,-63.775,-176.912,6.792,148.349
C04301=1209.597,262.847,-63.804,-176.909,6.795,148.349
C04302=1209.593,263.120,-63.835,-176.906,6.798,148.348
C04303=1209.588,263.392,-63.865,-176.903,6.800,148.348
C04304=1209.583,263.665,-63.895,-176.901,6.803,148.348
C04305=1209.578,263.914,-63.922,-176.898,6.805,148.348
C04306=1209.575,264.162,-63.950,-176.896,6.807,148.348
C04307=1209.570,264.411,-63.977,-176.893,6.810,148.347
C04308=1209.566,264.659,-64.005,-176.891,6.812,148.347
C04309=1209.561,264.907,-64.032,-176.888,6.814,148.347
C04310=1209.557,265.156,-64.060,-176.885,6.817,148.347
C04311=1209.553,265.404,-64.087,-176.883,6.819,148.347
C04312=1209.548,265.653,-64.114,-176.881,6.821,148.347
C04313=1209.544,265.901,-64.143,-176.878,6.824,148.347
C04314=1209.539,266.150,-64.170,-176.875,6.826,148.346
C04315=1209.534,266.398,-64.198,-176.873,6.828,148.346
C04316=1209.530,266.646,-64.225,-176.870,6.831,148.346
C04317=1209.526,266.895,-64.253,-176.868,6.833,148.346
C04318=1209.521,267.143,-64.280,-176.865,6.835,148.346
C04319=1209.517,267.391,-64.308,-176.863,6.838,148.345
C04320=1209.513,267.641,-64.335,-176.860,6.840,148.345
C04321=1209.509,267.888,-64.363,-176.858,6.842,148.345
C04322=1209.504,268.137,-64.390,-176.855,6.845,148.345
C04323=1209.499,268.386,-64.419,-176.853,6.847,148.345
C04324=1209.495,268.634,-64.446,-176.850,6.849,148.345
C04325=1209.490,268.882,-64.474,-176.847,6.852,148.344
C04326=1209.487,269.131,-64.502,-176.845,6.854,148.344
C04327=1209.482,269.379,-64.529,-176.843,6.856,148.344
C04328=1209.478,269.627,-64.557,-176.840,6.859,148.344
C04329=1209.473,269.877,-64.585,-176.838,6.861,148.344
C04330=1209.469,270.124,-64.613,-176.835,6.863,148.344
C04331=1209.464,270.372,-64.640,-176.832,6.866,148.344
C04332=1209.460,270.622,-64.668,-176.830,6.868,148.343
C04333=1209.456,270.869,-64.696,-176.828,6.870,148.343
C04334=1209.451,271.118,-64.724,-176.825,6.873,148.343
C04335=1209.447,271.366,-64.752,-176.822,6.875,148.343
C04336=1209.442,271.615,-64.779,-176.820,6.878,148.343
C04337=1209.439,271.863,-64.807,-176.817,6.880,148.343
C04338=1209.433,272.111,-64.836,-176.815,6.882,148.342
C04339=1209.429,272.361,-64.863,-176.812,6.885,148.342
C04340=1209.425,272.609,-64.891,-176.810,6.887,148.342
C04341=1209.420,272.857,-64.919,-176.807,6.889,148.342
C04342=1209.416,273.105,-64.947,-176.805,6.892,148.342
C04343=1209.412,273.353,-64.975,-176.802,6.894,148.342
C04344=1209.408,273.602,-65.003,-176.800,6.896,148.342
C04345=1209.403,273.851,-65.031,-176.797,6.899,148.341
C04346=1209.399,274.099,-65.059,-176.795,6.901,148.341
C04347=1209.395,274.347,-65.087,-176.792,6.904,148.341
C04348=1209.390,274.596,-65.116,-176.789,6.906,148.341
C04349=1209.386,274.844,-65.143,-176.787,6.908,148.341
C04350=1209.381,275.092,-65.172,-176.785,6.911,148.341
C04351=1209.377,275.341,-65.200,-176.782,6.913,148.341
C04352=1209.372,275.589,-65.227,-176.779,6.916,148.341
C04353=1209.368,275.838,-65.256,-176.777,6.918,148.341
C04354=1209.363,276.086,-65.284,-176.774,6.920,148.340
C04355=1209.360,276.334,-65.312,-176.772,6.923,148.340
C04356=1209.355,276.583,-65.340,-176.770,6.925,148.340
C04357=1209.351,276.831,-65.368,-176.767,6.927,148.340
C04358=1209.346,277.079,-65.397,-176.764,6.930,148.340
C04359=1209.342,277.328,-65.425,-176.762,6.932,148.340
C04360=1209.338,277.576,-65.452,-176.759,6.935,148.339
C04361=1209.333,277.825,-65.481,-176.757,6.937,148.339
C04362=1209.329,278.073,-65.509,-176.755,6.939,148.339
C04363=1209.324,278.321,-65.538,-176.752,6.942,148.339
C04364=1209.320,278.569,-65.566,-176.749,6.944,148.339
C04365=1209.315,278.818,-65.594,-176.747,6.947,148.339
C04366=1209.312,279.067,-65.622,-176.744,6.949,148.339
C04367=1209.307,279.314,-65.651,-176.742,6.952,148.339
C04368=1209.303,279.563,-65.680,-176.739,6.954,148.339
C04369=1209.298,279.811,-65.708,-176.737,6.956,148.338
C04370=1209.294,280.060,-65.736,-176.734,6.959,148.338
C04371=1209.289,280.308,-65.765,-176.732,6.961,148.338
C04372=1209.286,280.556,-65.793,-176.729,6.964,148.338
C04373=1209.280,280.805,-65.821,-176.727,6.966,148.338
C04374=1209.277,281.053,-65.850,-176.725,6.968,148.338
C04375=1209.273,281.301,-65.879,-176.722,6.971,148.338
C04376=1209.268,281.549,-65.906,-176.719,6.973,148.337
C04377=1209.264,281.798,-65.935,-176.717,6.976,148.337
C04378=1209.259,282.046,-65.964,-176.714,6.979,148.337
C04379=1209.255,282.294,-65.992,-176.711,6.981,148.337
C04380=1209.251,282.543,-66.021,-176.709,6.983,148.337
C04381=1209.246,282.791,-66.049,-176.707,6.986,148.337
C04382=1209.242,283.040,-66.078,-176.704,6.989,148.337
C04383=1209.237,283.288,-66.107,-176.702,6.991,148.337
C04384=1209.233,283.536,-66.135,-176.699,6.994,148.337
C04385=1209.229,283.785,-66.164,-176.697,6.996,148.337
C04386=1209.224,284.033,-66.193,-176.694,6.999,148.337
C04387=1209.220,284.281,-66.221,-176.692,7.001,148.336
C04388=1209.216,284.530,-66.250,-176.689,7.004,148.336
C04389=1209.212,284.777,-66.278,-176.687,7.006,148.336
C04390=1209.207,285.026,-66.307,-176.685,7.008,148.336
C04391=1209.202,285.274,-66.335,-176.681,7.011,148.336
C04392=1209.198,285.523,-66.365,-176.679,7.013,148.336
C04393=1209.194,285.771,-66.393,-176.677,7.016,148.336
C04394=1209.189,286.019,-66.421,-176.674,7.018,148.336
C04395=1209.185,286.268,-66.451,-176.671,7.021,148.335
C04396=1209.181,286.516,-66.479,-176.669,7.023,148.335
C04397=1209.177,286.765,-66.508,-176.667,7.026,148.335
C04398=1209.172,287.013,-66.537,-176.664,7.028,148.335
C04399=1209.168,287.261,-66.566,-176.661,7.031,148.335
C04400=1209.164,287.510,-66.594,-176.659,7.033,148.335
C04401=1209.159,287.757,-66.623,-176.657,7.035,148.335
C04402=1209.155,288.006,-66.652,-176.654,7.038,148.335
C04403=1209.151,288.254,-66.681,-176.652,7.041,148.335
C04404=1209.146,288.502,-66.709,-176.649,7.043,148.335
C04405=1209.141,288.776,-66.742,-176.646,7.046,148.335
C04406=1209.137,289.051,-66.774,-176.644,7.049,148.334
C04407=1209.132,289.326,-66.806,-176.641,7.051,148.334
C04408=1209.127,289.600,-66.837,-176.638,7.054,148.334
C04409=1209.122,289.848,-66.867,-176.636,7.057,148.334
C04410=1209.118,290.096,-66.896,-176.634,7.060,148.334
C04411=1209.114,290.344,-66.924,-176.631,7.063,148.334
C04412=1209.110,290.593,-66.954,-176.628,7.064,148.334
C04413=1209.105,290.840,-66.983,-176.626,7.067,148.334
C04414=1209.101,291.089,-67.011,-176.623,7.070,148.334
C04415=1209.097,291.337,-67.041,-176.621,7.073,148.334
C04416=1209.093,291.586,-67.070,-176.619,7.075,148.334
C04417=1209.088,291.835,-67.099,-176.616,7.077,148.334
C04418=1209.084,292.082,-67.128,-176.613,7.080,148.333
C04419=1209.080,292.330,-67.157,-176.611,7.082,148.333
C04420=1209.075,292.579,-67.186,-176.608,7.085,148.333
C04421=1209.071,292.827,-67.215,-176.606,7.087,148.333
C04422=1209.067,293.075,-67.245,-176.604,7.090,148.333
C04423=1209.062,293.323,-67.274,-176.602,7.092,148.333
C04424=1209.058,293.572,-67.302,-176.599,7.095,148.333
C04425=1209.054,293.820,-67.332,-176.596,7.097,148.333
C04426=1209.049,294.068,-67.361,-176.594,7.100,148.333
C04427=1209.045,294.317,-67.391,-176.591,7.103,148.333
C04428=1209.040,294.564,-67.420,-176.589,7.106,148.333
C04429=1209.036,294.813,-67.449,-176.587,7.108,148.333
C04430=1209.032,295.061,-67.478,-176.584,7.111,148.333
C04431=1209.028,295.310,-67.508,-176.582,7.113,148.333
C04432=1209.023,295.558,-67.537,-176.579,7.116,148.333
C04433=1209.019,295.806,-67.566,-176.577,7.118,148.333
C04434=1209.015,296.055,-67.596,-176.574,7.121,148.332
C04435=1209.010,296.302,-67.625,-176.572,7.123,148.332
C04436=1209.006,296.550,-67.654,-176.569,7.126,148.332
C04437=1209.002,296.799,-67.684,-176.567,7.128,148.332
C04438=1208.998,297.047,-67.713,-176.564,7.131,148.332
C04439=1208.994,297.295,-67.743,-176.562,7.134,148.332
C04440=1208.989,297.543,-67.772,-176.559,7.137,148.332
C04441=1208.985,297.792,-67.802,-176.557,7.139,148.332
C04442=1208.981,298.040,-67.831,-176.555,7.142,148.332
C04443=1208.977,298.288,-67.861,-176.552,7.145,148.332
C04444=1208.972,298.536,-67.890,-176.550,7.147,148.332
C04445=1208.968,298.784,-67.919,-176.547,7.150,148.332
C04446=1208.963,299.033,-67.949,-176.545,7.152,148.332
C04447=1208.959,299.281,-67.979,-176.542,7.155,148.332
C04448=1208.955,299.529,-68.008,-176.540,7.157,148.332
C04449=1208.950,299.777,-68.038,-176.537,7.160,148.331
C04450=1208.946,300.026,-68.067,-176.535,7.162,148.331
C04451=1208.942,300.274,-68.096,-176.532,7.165,148.331
C04452=1208.938,300.522,-68.126,-176.530,7.168,148.331
C04453=1208.933,300.771,-68.156,-176.527,7.171,148.331
C04454=1208.929,301.019,-68.185,-176.525,7.173,148.331
C04455=1208.925,301.267,-68.216,-176.523,7.176,148.331
C04456=1208.921,301.515,-68.245,-176.520,7.178,148.331
C04457=1208.917,301.763,-68.275,-176.518,7.181,148.331
C04458=1208.912,302.012,-68.304,-176.516,7.183,148.331
C04459=1208.907,302.260,-68.334,-176.513,7.186,148.331
C04460=1208.904,302.508,-68.364,-176.511,7.189,148.331
C04461=1208.899,302.756,-68.394,-176.508,7.192,148.331
C04462=1208.895,303.004,-68.423,-176.505,7.195,148.331
C04463=1208.890,303.253,-68.453,-176.503,7.197,148.331
C04464=1208.886,303.501,-68.483,-176.501,7.200,148.331
C04465=1208.882,303.749,-68.513,-176.499,7.202,148.331
C04466=1208.878,303.997,-68.542,-176.496,7.205,148.331
C04467=1208.873,304.246,-68.572,-176.494,7.207,148.331
C04468=1208.869,304.493,-68.602,-176.491,7.210,148.331
C04469=1208.865,304.742,-68.632,-176.489,7.213,148.331
C04470=1208.860,304.990,-68.662,-176.486,7.216,148.331
C04471=1208.856,305.238,-68.692,-176.484,7.218,148.331
C04472=1208.852,305.486,-68.722,-176.481,7.221,148.331
C04473=1208.847,305.735,-68.752,-176.479,7.224,148.331
C04474=1208.843,305.982,-68.782,-176.477,7.226,148.331
C04475=1208.839,306.231,-68.811,-176.474,7.229,148.331
C04476=1208.834,306.478,-68.842,-176.472,7.232,148.331
C04477=1208.830,306.727,-68.871,-176.470,7.235,148.331
C04478=1208.826,306.974,-68.902,-176.468,7.237,148.331
C04479=1208.821,307.223,-68.932,-176.465,7.240,148.331
C04480=1208.817,307.471,-68.961,-176.463,7.242,148.331
C04481=1208.813,307.719,-68.992,-176.460,7.245,148.331
C04482=1208.809,307.967,-69.021,-176.457,7.248,148.331
C04483=1208.805,308.215,-69.052,-176.455,7.250,148.331
C04484=1208.800,308.464,-69.082,-176.453,7.253,148.331
C04485=1208.796,308.712,-69.112,-176.450,7.256,148.330
C04486=1208.792,308.961,-69.142,-176.448,7.259,148.330
C04487=1208.788,309.208,-69.172,-176.446,7.261,148.330
C04488=1208.783,309.457,-69.202,-176.443,7.264,148.331
C04489=1208.779,309.705,-69.233,-176.441,7.266,148.331
C04490=1208.775,309.952,-69.263,-176.439,7.269,148.331
C04491=1208.770,310.201,-69.293,-176.436,7.272,148.331
C04492=1208.766,310.448,-69.323,-176.434,7.275,148.331
C04493=1208.762,310.698,-69.353,-176.431,7.278,148.331
C04494=1208.758,310.945,-69.383,-176.429,7.280,148.330
C04495=1208.753,311.193,-69.414,-176.426,7.283,148.330
C04496=1208.749,311.442,-69.444,-176.425,7.285,148.331
C04497=1208.745,311.689,-69.474,-176.422,7.288,148.331
C04498=1208.741,311.937,-69.505,-176.419,7.291,148.331
C04499=1208.736,312.186,-69.535,-176.417,7.294,148.331
C04500=1208.733,312.434,-69.565,-176.414,7.297,148.331
C04501=1208.728,312.682,-69.596,-176.412,7.299,148.330
C04502=1208.724,312.930,-69.626,-176.410,7.302,148.331
C04503=1208.719,313.178,-69.656,-176.408,7.304,148.331
C04504=1208.714,313.426,-69.687,-176.405,7.307,148.331
C04505=1208.711,313.675,-69.718,-176.403,7.310,148.331
C04506=1208.707,313.923,-69.748,-176.401,7.313,148.331
C04507=1208.702,314.171,-69.778,-176.398,7.316,148.331
C04508=1208.698,314.419,-69.808,-176.396,7.318,148.331
C04509=1208.693,314.695,-69.843,-176.394,7.321,148.331
C04510=1208.688,314.971,-69.876,-176.391,7.324,148.331
C04511=1208.684,315.246,-69.910,-176.388,7.327,148.331
C04512=1208.679,315.524,-69.944,-176.386,7.330,148.331
C04513=1208.675,315.771,-69.975,-176.383,7.333,148.331
C04514=1208.670,316.019,-70.005,-176.381,7.336,148.331
C04515=1208.666,316.267,-70.036,-176.378,7.339,148.331
C04516=1208.662,316.516,-70.067,-176.376,7.342,148.331
C04517=1208.658,316.764,-70.098,-176.374,7.344,148.331
C04518=1208.654,317.011,-70.128,-176.371,7.348,148.331
C04519=1208.649,317.259,-70.158,-176.369,7.350,148.331
C04520=1208.645,317.508,-70.190,-176.367,7.353,148.331
C04521=1208.641,317.756,-70.220,-176.365,7.355,148.331
C04522=1208.637,318.004,-70.251,-176.362,7.358,148.331
C04523=1208.632,318.252,-70.281,-176.360,7.361,148.331
C04524=1208.629,318.500,-70.312,-176.358,7.364,148.331
C04525=1208.624,318.748,-70.343,-176.355,7.367,148.331
C04526=1208.620,318.996,-70.373,-176.353,7.369,148.331
C04527=1208.616,319.244,-70.404,-176.351,7.372,148.331
C04528=1208.612,319.492,-70.435,-176.348,7.375,148.331
C04529=1208.607,319.740,-70.465,-176.346,7.378,148.331
C04530=1208.603,319.989,-70.497,-176.344,7.381,148.331
C04531=1208.598,320.237,-70.527,-176.341,7.383,148.331
C04532=1208.594,320.485,-70.558,-176.339,7.386,148.332
C04533=1208.591,320.733,-70.589,-176.337,7.389,148.332
C04534=1208.586,320.981,-70.619,-176.334,7.392,148.332
C04535=1208.581,321.229,-70.650,-176.332,7.395,148.332
C04536=1208.578,321.477,-70.682,-176.330,7.397,148.332
C04537=1208.573,321.725,-70.713,-176.327,7.400,148.332
C04538=1208.569,321.973,-70.743,-176.326,7.403,148.332
C04539=1208.565,322.221,-70.774,-176.323,7.406,148.332
C04540=1208.561,322.469,-70.805,-176.320,7.409,148.332
C04541=1208.556,322.717,-70.836,-176.319,7.411,148.332
C04542=1208.552,322.965,-70.867,-176.316,7.414,148.332
C04543=1208.548,323.213,-70.898,-176.314,7.416,148.332
C04544=1208.544,323.461,-70.928,-176.312,7.420,148.332
C04545=1208.540,323.709,-70.959,-176.309,7.423,148.332
C04546=1208.535,323.957,-70.991,-176.307,7.425,148.332
C04547=1208.531,324.205,-71.022,-176.305,7.428,148.332
C04548=1208.527,324.453,-71.053,-176.303,7.431,148.332
C04549=1208.522,324.701,-71.084,-176.300,7.434,148.333
C04550=1208.518,324.949,-71.115,-176.298,7.437,148.333
C04551=1208.514,325.197,-71.146,-176.296,7.439,148.333
C04552=1208.510,325.446,-71.177,-176.293,7.443,148.333
C04553=1208.506,325.693,-71.209,-176.292,7.445,148.333
C04554=1208.502,325.942,-71.240,-176.289,7.448,148.333
C04555=1208.498,326.189,-71.271,-176.286,7.451,148.333
C04556=1208.493,326.437,-71.302,-176.285,7.454,148.333
C04557=1208.489,326.686,-71.333,-176.282,7.457,148.333
C04558=1208.485,326.933,-71.364,-176.280,7.459,148.333
C04559=1208.481,327.182,-71.395,-176.278,7.462,148.333
C04560=1208.477,327.429,-71.427,-176.275,7.466,148.333
C04561=1208.473,327.678,-71.458,-176.273,7.468,148.333
C04562=1208.468,327.926,-71.489,-176.271,7.471,148.334
C04563=1208.464,328.174,-71.521,-176.269,7.473,148.334
C04564=1208.460,328.422,-71.551,-176.267,7.477,148.334
C04565=1208.455,328.670,-71.584,-176.264,7.480,148.334
C04566=1208.451,328.918,-71.615,-176.263,7.482,148.334
C04567=1208.446,329.165,-71.646,-176.260,7.485,148.334
C04568=1208.442,329.414,-71.677,-176.258,7.488,148.334
C04569=1208.438,329.661,-71.709,-176.255,7.491,148.334
C04570=1208.434,329.910,-71.740,-176.253,7.494,148.334
C04571=1208.430,330.157,-71.771,-176.251,7.496,148.334
C04572=1208.426,330.405,-71.803,-176.249,7.500,148.335
C04573=1208.421,330.653,-71.834,-176.247,7.502,148.334
C04574=1208.418,330.901,-71.866,-176.245,7.505,148.335
C04575=1208.413,331.149,-71.896,-176.242,7.509,148.335
C04576=1208.409,331.397,-71.928,-176.240,7.511,148.335
C04577=1208.405,331.646,-71.961,-176.238,7.514,148.335
C04578=1208.400,331.894,-71.992,-176.236,7.516,148.335
C04579=1208.397,332.142,-72.023,-176.234,7.520,148.335
C04580=1208.392,332.389,-72.055,-176.232,7.522,148.335
C04581=1208.388,332.638,-72.086,-176.229,7.525,148.335
C04582=1208.384,332.885,-72.117,-176.227,7.529,148.336
C04583=1208.380,333.133,-72.150,-176.225,7.531,148.336
C04584=1208.375,333.381,-72.181,-176.223,7.534,148.336
C04585=1208.371,333.629,-72.212,-176.221,7.537,148.336
C04586=1208.367,333.877,-72.244,-176.219,7.540,148.336
C04587=1208.363,334.125,-72.276,-176.216,7.543,148.336
C04588=1208.358,334.374,-72.308,-176.214,7.545,148.336
C04589=1208.354,334.621,-72.339,-176.212,7.549,148.336
C04590=1208.350,334.869,-72.371,-176.210,7.551,148.337
C04591=1208.346,335.116,-72.402,-176.208,7.554,148.337
C04592=1208.342,335.364,-72.434,-176.205,7.557,148.337
C04593=1208.338,335.613,-72.466,-176.204,7.560,148.337
C04594=1208.333,335.861,-72.497,-176.201,7.563,148.337
C04595=1208.330,336.109,-72.529,-176.199,7.566,148.337
C04596=1208.325,336.356,-72.561,-176.197,7.569,148.337
C04597=1208.321,336.604,-72.593,-176.195,7.572,148.338
C04598=1208.317,336.852,-72.625,-176.193,7.574,148.338
C04599=1208.313,337.100,-72.656,-176.191,7.578,148.338
C04600=1208.308,337.349,-72.688,-176.189,7.580,148.338
C04601=1208.304,337.597,-72.720,-176.186,7.583,148.338
C04602=1208.300,337.844,-72.752,-176.185,7.586,148.338
C04603=1208.296,338.092,-72.784,-176.183,7.589,148.338
C04604=1208.291,338.340,-72.815,-176.180,7.593,148.339
C04605=1208.288,338.588,-72.847,-176.178,7.595,148.339
C04606=1208.283,338.836,-72.880,-176.176,7.598,148.339
C04607=1208.279,339.084,-72.911,-176.174,7.601,148.339
C04608=1208.275,339.332,-72.943,-176.172,7.604,148.339
C04609=1208.271,339.580,-72.976,-176.169,7.607,148.339
C04610=1208.266,339.827,-73.007,-176.168,7.609,148.339
C04611=1208.263,340.075,-73.039,-176.166,7.613,148.340
C04612=1208.258,340.324,-73.071,-176.164,7.615,148.340
C04613=1208.254,340.601,-73.107,-176.162,7.619,148.340
C04614=1208.249,340.879,-73.143,-176.159,7.622,148.340
C04615=1208.244,341.158,-73.179,-176.157,7.625,148.340
C04616=1208.239,341.436,-73.215,-176.155,7.628,148.340
C04617=1208.235,341.684,-73.247,-176.152,7.632,148.341
C04618=1208.232,341.932,-73.279,-176.150,7.635,148.341
C04619=1208.227,342.180,-73.311,-176.149,7.638,148.341
C04620=1208.223,342.427,-73.343,-176.146,7.641,148.341
C04621=1208.219,342.676,-73.376,-176.144,7.643,148.341
C04622=1208.215,342.923,-73.407,-176.142,7.647,148.341
C04623=1208.210,343.171,-73.440,-176.140,7.649,148.342
C04624=1208.206,343.419,-73.472,-176.138,7.652,148.342
C04625=1208.202,343.668,-73.504,-176.136,7.656,148.342
C04626=1208.198,343.914,-73.536,-176.134,7.658,148.342
C04627=1208.193,344.163,-73.569,-176.132,7.662,148.343
C04628=1208.190,344.411,-73.601,-176.130,7.664,148.343
C04629=1208.185,344.659,-73.633,-176.128,7.667,148.343
C04630=1208.181,344.906,-73.665,-176.127,7.670,148.343
C04631=1208.177,345.154,-73.698,-176.124,7.673,148.343
C04632=1208.173,345.402,-73.730,-176.122,7.676,148.343
C04633=1208.169,345.651,-73.762,-176.120,7.679,148.344
C04634=1208.164,345.898,-73.795,-176.118,7.682,148.344
C04635=1208.160,346.146,-73.827,-176.116,7.685,148.344
C04636=1208.156,346.394,-73.859,-176.114,7.688,148.344
C04637=1208.152,346.641,-73.892,-176.112,7.691,148.344
C04638=1208.148,346.890,-73.924,-176.110,7.694,148.345
C04639=1208.143,347.137,-73.956,-176.108,7.697,148.345
C04640=1208.140,347.385,-73.989,-176.106,7.700,148.345
C04641=1208.135,347.633,-74.021,-176.104,7.703,148.345
C04642=1208.132,347.881,-74.054,-176.102,7.706,148.345
C04643=1208.127,348.129,-74.086,-176.101,7.709,148.346
C04644=1208.122,348.377,-74.118,-176.099,7.712,148.346
C04645=1208.119,348.624,-74.151,-176.097,7.715,148.346
C04646=1208.114,348.872,-74.183,-176.095,7.718,148.346
C04647=1208.110,349.120,-74.216,-176.093,7.721,148.347
C04648=1208.107,349.368,-74.248,-176.091,7.724,148.347
C04649=1208.102,349.616,-74.281,-176.089,7.727,148.347
C04650=1208.097,349.863,-74.313,-176.087,7.730,148.347
C04651=1208.094,350.111,-74.346,-176.085,7.733,148.347
C04652=1208.090,350.359,-74.378,-176.083,7.736,148.348
C04653=1208.085,350.607,-74.412,-176.081,7.739,148.348
C04654=1208.082,350.855,-74.443,-176.080,7.742,148.348
C04655=1208.078,351.103,-74.477,-176.078,7.745,148.348
C04656=1208.073,351.351,-74.509,-176.076,7.748,148.349
C04657=1208.069,351.599,-74.542,-176.074,7.751,148.349
C04658=1208.065,351.846,-74.574,-176.072,7.754,148.349
C04659=1208.061,352.094,-74.607,-176.070,7.757,148.349
C04660=1208.056,352.342,-74.640,-176.068,7.760,148.349
C04661=1208.053,352.590,-74.672,-176.066,7.763,148.350
C04662=1208.049,352.837,-74.705,-176.065,7.766,148.350
C04663=1208.044,353.085,-74.738,-176.062,7.769,148.350
C04664=1208.040,353.333,-74.771,-176.061,7.772,148.350
C04665=1208.036,353.581,-74.804,-176.059,7.775,148.351
C04666=1208.032,353.829,-74.836,-176.057,7.778,148.351
C04667=1208.028,354.077,-74.869,-176.055,7.781,148.351
C04668=1208.023,354.324,-74.901,-176.053,7.784,148.352
C04669=1208.019,354.572,-74.935,-176.052,7.787,148.352
C04670=1208.015,354.820,-74.967,-176.050,7.790,148.352
C04671=1208.011,355.067,-75.000,-176.048,7.793,148.352
C04672=1208.007,355.315,-75.033,-176.046,7.796,148.353
C04673=1208.003,355.564,-75.065,-176.044,7.799,148.353
C04674=1207.999,355.811,-75.098,-176.043,7.802,148.353
C04675=1207.994,356.059,-75.132,-176.040,7.805,148.353
C04676=1207.990,356.307,-75.165,-176.039,7.808,148.354
C04677=1207.987,356.554,-75.197,-176.037,7.811,148.354
C04678=1207.982,356.803,-75.230,-176.035,7.814,148.354
C04679=1207.978,357.050,-75.263,-176.034,7.818,148.355
C04680=1207.974,357.298,-75.296,-176.031,7.821,148.355
C04681=1207.970,357.546,-75.329,-176.030,7.823,148.355
C04682=1207.966,357.793,-75.362,-176.028,7.827,148.355
C04683=1207.961,358.042,-75.395,-176.026,7.830,148.356
C04684=1207.957,358.290,-75.428,-176.025,7.833,148.356
C04685=1207.953,358.537,-75.461,-176.023,7.836,148.356
C04686=1207.949,358.785,-75.494,-176.021,7.839,148.357
C04687=1207.946,359.032,-75.527,-176.020,7.842,148.357
C04688=1207.941,359.280,-75.560,-176.018,7.844,148.357
C04689=1207.937,359.528,-75.593,-176.016,7.848,148.358
C04690=1207.933,359.776,-75.626,-176.014,7.851,148.358
C04691=1207.929,360.023,-75.659,-176.013,7.854,148.358
C04692=1207.925,360.271,-75.693,-176.011,7.857,148.358
C04693=1207.921,360.519,-75.726,-176.009,7.860,148.359
C04694=1207.917,360.767,-75.759,-176.008,7.863,148.359
C04695=1207.912,361.014,-75.792,-176.006,7.867,148.359
C04696=1207.908,361.262,-75.825,-176.004,7.869,148.360
C04697=1207.904,361.510,-75.858,-176.002,7.873,148.360
C04698=1207.900,361.757,-75.892,-176.001,7.875,148.360
C04699=1207.896,362.005,-75.925,-175.999,7.879,148.361
C04700=1207.892,362.253,-75.958,-175.997,7.881,148.361
C04701=1207.888,362.501,-75.991,-175.996,7.884,148.361
C04702=1207.884,362.748,-76.024,-175.994,7.888,148.361
C04703=1207.880,362.997,-76.058,-175.993,7.890,148.362
C04704=1207.876,363.245,-76.091,-175.991,7.894,148.362
C04705=1207.872,363.492,-76.124,-175.989,7.897,148.362
C04706=1207.868,363.740,-76.157,-175.988,7.900,148.363
C04707=1207.863,363.988,-76.190,-175.986,7.903,148.363
C04708=1207.859,364.235,-76.223,-175.985,7.906,148.363
C04709=1207.855,364.483,-76.258,-175.983,7.909,148.364
C04710=1207.851,364.731,-76.291,-175.982,7.912,148.364
C04711=1207.846,364.978,-76.324,-175.980,7.915,148.365
C04712=1207.842,365.226,-76.357,-175.978,7.918,148.365
C04713=1207.838,365.474,-76.391,-175.977,7.921,148.365
C04714=1207.835,365.722,-76.424,-175.975,7.924,148.366
C04715=1207.831,365.969,-76.458,-175.974,7.927,148.366
C04716=1207.827,366.217,-76.491,-175.973,7.930,148.366
C04717=1207.822,366.498,-76.530,-175.971,7.934,148.367
C04718=1207.817,366.778,-76.566,-175.969,7.937,148.367
C04719=1207.812,367.058,-76.605,-175.967,7.941,148.367
C04720=1207.808,367.339,-76.643,-175.965,7.944,148.368
C04721=1207.804,367.586,-76.676,-175.964,7.947,148.368
C04722=1207.800,367.834,-76.709,-175.963,7.950,148.369
C04723=1207.795,368.082,-76.744,-175.961,7.953,148.369
C04724=1207.791,368.329,-76.777,-175.960,7.956,148.370
C04725=1207.787,368.577,-76.810,-175.958,7.959,148.370
C04726=1207.783,368.825,-76.843,-175.957,7.962,148.370
C04727=1207.780,369.073,-76.877,-175.955,7.965,148.371
C04728=1207.775,369.321,-76.911,-175.954,7.968,148.371
C04729=1207.771,369.568,-76.944,-175.953,7.971,148.371
C04730=1207.767,369.815,-76.978,-175.951,7.975,148.372
C04731=1207.763,370.063,-77.011,-175.950,7.977,148.372
C04732=1207.759,370.310,-77.045,-175.949,7.980,148.373
C04733=1207.755,370.559,-77.079,-175.947,7.983,148.373
C04734=1207.751,370.807,-77.112,-175.945,7.986,148.373
C04735=1207.747,371.054,-77.146,-175.944,7.989,148.374
C04736=1207.743,371.302,-77.179,-175.943,7.992,148.374
C04737=1207.738,371.549,-77.214,-175.942,7.995,148.374
C04738=1207.734,371.797,-77.247,-175.940,7.998,148.375
C04739=1207.730,372.045,-77.281,-175.939,8.001,148.375
C04740=1207.727,372.292,-77.314,-175.937,8.004,148.376
C04741=1207.722,372.540,-77.348,-175.936,8.007,148.376
C04742=1207.718,372.787,-77.382,-175.935,8.010,148.376
C04743=1207.714,373.036,-77.416,-175.933,8.013,148.377
C04744=1207.710,373.283,-77.450,-175.932,8.016,148.377
C04745=1207.706,373.531,-77.483,-175.931,8.019,148.378
C04746=1207.702,373.778,-77.517,-175.930,8.022,148.378
C04747=1207.697,374.027,-77.551,-175.929,8.025,148.379
C04748=1207.694,374.274,-77.585,-175.928,8.028,148.379
C04749=1207.689,374.522,-77.618,-175.926,8.031,148.379
C04750=1207.685,374.769,-77.653,-175.925,8.034,148.380
C04751=1207.681,375.018,-77.686,-175.923,8.037,148.380
C04752=1207.678,375.265,-77.720,-175.922,8.040,148.381
C04753=1207.673,375.512,-77.754,-175.921,8.043,148.381
C04754=1207.669,375.760,-77.788,-175.920,8.046,148.382
C04755=1207.666,376.008,-77.822,-175.919,8.048,148.382
C04756=1207.661,376.256,-77.856,-175.918,8.051,148.382
C04757=1207.657,376.503,-77.890,-175.916,8.055,148.383
C04758=1207.653,376.751,-77.923,-175.915,8.058,148.383
C04759=1207.649,376.999,-77.957,-175.914,8.061,148.384
C04760=1207.645,377.246,-77.991,-175.913,8.064,148.384
C04761=1207.640,377.494,-78.025,-175.912,8.066,148.385
C04762=1207.636,377.741,-78.059,-175.911,8.069,148.385
C04763=1207.633,377.989,-78.093,-175.909,8.072,148.385
C04764=1207.628,378.237,-78.127,-175.909,8.075,148.386
C04765=1207.624,378.484,-78.161,-175.907,8.078,148.386
C04766=1207.620,378.732,-78.196,-175.906,8.081,148.387
C04767=1207.616,378.980,-78.229,-175.905,8.084,148.387
C04768=1207.612,379.227,-78.263,-175.904,8.087,148.388
C04769=1207.608,379.474,-78.297,-175.903,8.089,148.388
C04770=1207.604,379.722,-78.332,-175.902,8.092,148.388
C04771=1207.600,379.970,-78.365,-175.901,8.095,148.389
C04772=1207.596,380.217,-78.399,-175.900,8.098,148.389
C04773=1207.592,380.465,-78.434,-175.899,8.101,148.390
C04774=1207.588,380.713,-78.467,-175.898,8.104,148.390
C04775=1207.583,380.960,-78.501,-175.897,8.107,148.391
C04776=1207.580,381.208,-78.536,-175.895,8.110,148.391
C04777=1207.575,381.456,-78.570,-175.895,8.113,148.392
C04778=1207.572,381.703,-78.604,-175.893,8.116,148.392
C04779=1207.567,381.952,-78.638,-175.892,8.118,148.393
C04780=1207.563,382.199,-78.672,-175.892,8.121,148.393
C04781=1207.559,382.446,-78.707,-175.891,8.124,148.394
C04782=1207.556,382.694,-78.741,-175.890,8.127,148.394
C04783=1207.551,382.941,-78.775,-175.889,8.129,148.394
C04784=1207.547,383.189,-78.808,-175.888,8.133,148.395
C04785=1207.543,383.437,-78.843,-175.887,8.135,148.395
C04786=1207.538,383.685,-78.878,-175.886,8.138,148.396
C04787=1207.535,383.932,-78.912,-175.885,8.141,148.396
C04788=1207.531,384.180,-78.946,-175.884,8.143,148.397
C04789=1207.527,384.427,-78.980,-175.884,8.146,148.397
C04790=1207.523,384.675,-79.015,-175.882,8.149,148.398
C04791=1207.519,384.922,-79.049,-175.882,8.152,148.398
C04792=1207.514,385.170,-79.083,-175.880,8.155,148.399
C04793=1207.511,385.418,-79.117,-175.880,8.158,148.399
C04794=1207.506,385.665,-79.151,-175.879,8.160,148.400
C04795=1207.502,385.913,-79.186,-175.878,8.163,148.400
C04796=1207.498,386.161,-79.220,-175.877,8.166,148.401
C04797=1207.494,386.408,-79.255,-175.876,8.169,148.401
C04798=1207.491,386.656,-79.289,-175.876,8.171,148.402
C04799=1207.486,386.903,-79.323,-175.875,8.174,148.402
C04800=1207.482,387.151,-79.358,-175.874,8.177,148.403
C04801=1207.478,387.399,-79.392,-175.873,8.180,148.403
C04802=1207.474,387.646,-79.426,-175.873,8.182,148.404
C04803=1207.471,387.894,-79.461,-175.871,8.185,148.404
C04804=1207.466,388.141,-79.495,-175.871,8.188,148.405
C04805=1207.461,388.389,-79.530,-175.870,8.190,148.405
C04806=1207.458,388.636,-79.564,-175.869,8.193,148.406
C04807=1207.454,388.884,-79.598,-175.868,8.196,148.406
C04808=1207.450,389.132,-79.633,-175.867,8.199,148.407
C04809=1207.446,389.379,-79.667,-175.867,8.202,148.407
C04810=1207.442,389.627,-79.702,-175.866,8.204,148.408
C04811=1207.438,389.874,-79.736,-175.866,8.207,148.408
C04812=1207.433,390.122,-79.770,-175.864,8.210,148.408
C04813=1207.429,390.370,-79.805,-175.864,8.213,148.409
C04814=1207.426,390.617,-79.839,-175.863,8.215,148.410
C04815=1207.422,390.865,-79.874,-175.862,8.218,148.410
C04816=1207.417,391.112,-79.908,-175.861,8.221,148.411
C04817=1207.414,391.360,-79.942,-175.861,8.223,148.411
C04818=1207.410,391.607,-79.978,-175.860,8.226,148.412
C04819=1207.405,391.855,-80.012,-175.860,8.228,148.412
C04820=1207.402,392.102,-80.046,-175.859,8.231,148.413
C04821=1207.397,392.385,-80.085,-175.858,8.234,148.413
C04822=1207.392,392.667,-80.125,-175.857,8.237,148.414
C04823=1207.387,392.950,-80.165,-175.856,8.240,148.414
C04824=1207.383,393.233,-80.204,-175.856,8.243,148.415
C04825=1207.379,393.480,-80.238,-175.855,8.246,148.415
C04826=1207.375,393.728,-80.273,-175.855,8.249,148.416
C04827=1207.370,393.975,-80.308,-175.854,8.251,148.416
C04828=1207.367,394.222,-80.343,-175.853,8.254,148.417
C04829=1207.363,394.470,-80.377,-175.853,8.256,148.417
C04830=1207.359,394.718,-80.412,-175.852,8.258,148.418
C04831=1207.354,394.965,-80.446,-175.852,8.261,148.418
C04832=1207.351,395.213,-80.481,-175.851,8.264,148.419
C04833=1207.347,395.461,-80.515,-175.850,8.266,148.419
C04834=1207.343,395.708,-80.551,-175.850,8.269,148.420
C04835=1207.338,395.956,-80.585,-175.849,8.272,148.420
C04836=1207.335,396.203,-80.619,-175.849,8.274,148.421
C04837=1207.330,396.451,-80.654,-175.848,8.277,148.421
C04838=1207.327,396.698,-80.689,-175.848,8.279,148.422
C04839=1207.322,396.946,-80.724,-175.847,8.281,148.422
C04840=1207.318,397.194,-80.759,-175.846,8.284,148.423
C04841=1207.314,397.441,-80.792,-175.846,8.286,148.423
C04842=1207.311,397.688,-80.828,-175.845,8.289,148.424
C04843=1207.306,397.936,-80.862,-175.845,8.292,148.424
C04844=1207.302,398.184,-80.897,-175.844,8.294,148.425
C04845=1207.298,398.431,-80.932,-175.843,8.297,148.425
C04846=1207.295,398.679,-80.967,-175.843,8.299,148.426
C04847=1207.290,398.926,-81.001,-175.843,8.301,148.426
C04848=1207.286,399.174,-81.036,-175.842,8.304,148.427
C04849=1207.282,399.422,-81.070,-175.842,8.306,148.427
C04850=1207.278,399.669,-81.106,-175.841,8.309,148.428
C04851=1207.274,399.916,-81.140,-175.840,8.312,148.428
C04852=1207.270,400.164,-81.175,-175.840,8.314,148.429
C04853=1207.266,400.411,-81.210,-175.840,8.316,148.429
C04854=1207.262,400.659,-81.245,-175.839,8.319,148.430
C04855=1207.257,400.907,-81.279,-175.838,8.321,148.430
C04856=1207.254,401.154,-81.315,-175.838,8.323,148.431
C04857=1207.250,401.401,-81.349,-175.838,8.326,148.431
C04858=1207.246,401.649,-81.383,-175.837,8.329,148.432
C04859=1207.242,401.896,-81.419,-175.836,8.331,148.432
C04860=1207.238,402.144,-81.453,-175.836,8.333,148.433
C04861=1207.234,402.392,-81.489,-175.836,8.335,148.433
C04862=1207.229,402.639,-81.523,-175.835,8.338,148.434
C04863=1207.225,402.887,-81.558,-175.835,8.340,148.434
C04864=1207.222,403.134,-81.593,-175.834,8.343,148.435
C04865=1207.218,403.382,-81.628,-175.834,8.345,148.435
C04866=1207.214,403.629,-81.663,-175.833,8.348,148.436
C04867=1207.210,403.877,-81.698,-175.833,8.350,148.436
C04868=1207.205,404.124,-81.732,-175.833,8.352,148.437
C04869=1207.202,404.372,-81.768,-175.832,8.355,148.437
C04870=1207.198,404.620,-81.803,-175.832,8.357,148.438
C04871=1207.193,404.867,-81.838,-175.831,8.359,148.438
C04872=1207.189,405.115,-81.873,-175.831,8.362,148.439
C04873=1207.185,405.362,-81.906,-175.830,8.364,148.439
C04874=1207.182,405.609,-81.942,-175.830,8.366,148.440
C04875=1207.177,405.857,-81.976,-175.830,8.368,148.440
C04876=1207.174,406.104,-82.012,-175.829,8.371,148.441
C04877=1207.170,406.352,-82.047,-175.829,8.373,148.441
C04878=1207.165,406.599,-82.082,-175.828,8.376,148.442
C04879=1207.161,406.847,-82.117,-175.828,8.378,148.442
C04880=1207.157,407.094,-82.152,-175.828,8.380,148.443
C04881=1207.153,407.342,-82.187,-175.827,8.383,148.443
C04882=1207.149,407.590,-82.222,-175.827,8.385,148.444
C04883=1207.145,407.837,-82.257,-175.826,8.387,148.444
C04884=1207.141,408.085,-82.292,-175.826,8.389,148.445
C04885=1207.137,408.332,-82.327,-175.826,8.391,148.445
C04886=1207.134,408.579,-82.362,-175.825,8.393,148.446
C04887=1207.130,408.827,-82.397,-175.825,8.396,148.446
C04888=1207.126,409.074,-82.432,-175.824,8.399,148.447
C04889=1207.122,409.322,-82.467,-175.824,8.401,148.447
C04890=1207.117,409.569,-82.502,-175.823,8.403,148.448
C04891=1207.113,409.817,-82.537,-175.823,8.405,148.448
C04892=1207.110,410.065,-82.572,-175.823,8.407,148.449
C04893=1207.105,410.312,-82.607,-175.822,8.409,148.449
C04894=1207.101,410.560,-82.642,-175.822,8.412,148.450
C04895=1207.097,410.806,-82.677,-175.822,8.414,148.450
C04896=1207.093,411.055,-82.712,-175.822,8.416,148.451
C04897=1207.090,411.302,-82.748,-175.821,8.418,148.451
C04898=1207.085,411.549,-82.782,-175.821,8.420,148.451
C04899=1207.081,411.797,-82.818,-175.821,8.423,148.452
C04900=1207.077,412.045,-82.853,-175.820,8.425,148.452
C04901=1207.073,412.292,-82.888,-175.820,8.427,148.453
C04902=1207.069,412.539,-82.923,-175.820,8.429,148.453
C04903=1207.065,412.787,-82.958,-175.819,8.431,148.454
C04904=1207.061,413.034,-82.993,-175.819,8.433,148.454
C04905=1207.057,413.282,-83.028,-175.818,8.436,148.455
C04906=1207.053,413.529,-83.063,-175.818,8.438,148.455
C04907=1207.049,413.777,-83.099,-175.818,8.440,148.456
C04908=1207.045,414.025,-83.134,-175.817,8.442,148.456
C04909=1207.041,414.272,-83.169,-175.817,8.444,148.457
C04910=1207.037,414.519,-83.205,-175.816,8.446,148.457
C04911=1207.033,414.767,-83.239,-175.816,8.449,148.458
C04912=1207.029,415.014,-83.275,-175.816,8.451,148.458
C04913=1207.025,415.262,-83.310,-175.815,8.453,148.458
C04914=1207.021,415.509,-83.345,-175.815,8.455,148.459
C04915=1207.017,415.757,-83.380,-175.815,8.457,148.459
C04916=1207.014,416.004,-83.416,-175.815,8.459,148.460
C04917=1207.008,416.277,-83.454,-175.814,8.462,148.460
C04918=1207.004,416.550,-83.493,-175.814,8.464,148.461
C04919=1207.003,416.823,-83.532,-175.814,8.466,148.461
C04920=1207.005,417.095,-83.570,-175.813,8.468,148.462
C04921=1206.584,417.095,-83.607,-175.816,8.479,148.465
C04922=1206.581,416.820,-83.568,-175.816,8.477,148.465
C04923=1206.583,416.544,-83.530,-175.817,8.475,148.465
C04924=1206.587,416.269,-83.490,-175.817,8.472,148.464
C04925=1206.592,415.994,-83.451,-175.818,8.469,148.463
C04926=1206.595,415.746,-83.416,-175.818,8.467,148.463
C04927=1206.599,415.498,-83.381,-175.818,8.466,148.463
C04928=1206.603,415.251,-83.346,-175.819,8.464,148.462
C04929=1206.607,415.004,-83.310,-175.819,8.461,148.462
C04930=1206.611,414.756,-83.275,-175.819,8.459,148.461
C04931=1206.615,414.509,-83.240,-175.820,8.457,148.461
C04932=1206.619,414.262,-83.205,-175.820,8.455,148.460
C04933=1206.624,414.013,-83.169,-175.821,8.453,148.460
C04934=1206.628,413.766,-83.134,-175.821,8.451,148.459
C04935=1206.632,413.518,-83.099,-175.821,8.448,148.459
C04936=1206.636,413.271,-83.064,-175.822,8.446,148.458
C04937=1206.640,413.024,-83.028,-175.822,8.444,148.458
C04938=1206.644,412.776,-82.994,-175.822,8.442,148.457
C04939=1206.647,412.528,-82.958,-175.822,8.440,148.457
C04940=1206.652,412.281,-82.923,-175.823,8.438,148.457
C04941=1206.656,412.033,-82.888,-175.823,8.435,148.456
C04942=1206.660,411.787,-82.853,-175.823,8.433,148.455
C04943=1206.664,411.538,-82.818,-175.824,8.431,148.455
C04944=1206.668,411.291,-82.783,-175.824,8.429,148.455
C04945=1206.672,411.044,-82.747,-175.825,8.427,148.454
C04946=1206.676,410.796,-82.713,-175.825,8.424,148.454
C04947=1206.680,410.549,-82.677,-175.825,8.422,148.453
C04948=1206.683,410.301,-82.643,-175.826,8.420,148.453
C04949=1206.687,410.054,-82.608,-175.826,8.418,148.452
C04950=1206.692,409.806,-82.573,-175.827,8.416,148.452
C04951=1206.695,409.559,-82.538,-175.827,8.414,148.451
C04952=1206.699,409.311,-82.503,-175.827,8.411,148.451
C04953=1206.703,409.064,-82.468,-175.827,8.409,148.450
C04954=1206.707,408.817,-82.432,-175.828,8.407,148.450
C04955=1206.712,408.569,-82.398,-175.829,8.404,148.449
C04956=1206.715,408.322,-82.362,-175.829,8.402,148.449
C04957=1206.719,408.074,-82.327,-175.829,8.399,148.448
C04958=1206.724,407.827,-82.292,-175.830,8.397,148.448
C04959=1206.728,407.579,-82.257,-175.830,8.395,148.447
C04960=1206.732,407.332,-82.222,-175.830,8.393,148.447
C04961=1206.736,407.084,-82.187,-175.830,8.391,148.446
C04962=1206.739,406.836,-82.152,-175.831,8.389,148.446
C04963=1206.744,406.589,-82.117,-175.831,8.386,148.445
C04964=1206.748,406.341,-82.082,-175.831,8.384,148.445
C04965=1206.752,406.094,-82.047,-175.832,8.381,148.444
C04966=1206.755,405.846,-82.013,-175.833,8.379,148.444
C04967=1206.759,405.599,-81.977,-175.833,8.377,148.443
C04968=1206.764,405.351,-81.943,-175.833,8.375,148.443
C04969=1206.767,405.104,-81.907,-175.834,8.372,148.442
C04970=1206.772,404.856,-81.873,-175.834,8.370,148.442
C04971=1206.776,404.609,-81.837,-175.834,8.368,148.442
C04972=1206.780,404.361,-81.803,-175.835,8.365,148.441
C04973=1206.784,404.114,-81.767,-175.835,8.363,148.440
C04974=1206.788,403.866,-81.732,-175.836,8.361,148.440
C04975=1206.792,403.618,-81.698,-175.836,8.358,148.440
C04976=1206.795,403.371,-81.663,-175.837,8.356,148.439
C04977=1206.800,403.124,-81.629,-175.837,8.353,148.438
C04978=1206.804,402.876,-81.593,-175.838,8.351,148.438
C04979=1206.808,402.629,-81.559,-175.838,8.349,148.438
C04980=1206.812,402.381,-81.524,-175.838,8.346,148.437
C04981=1206.816,402.134,-81.489,-175.839,8.343,148.436
C04982=1206.820,401.886,-81.454,-175.840,8.341,148.436
C04983=1206.824,401.638,-81.418,-175.840,8.339,148.436
C04984=1206.828,401.391,-81.384,-175.840,8.337,148.435
C04985=1206.832,401.143,-81.349,-175.841,8.334,148.434
C04986=1206.836,400.896,-81.314,-175.842,8.332,148.434
C04987=1206.840,400.648,-81.279,-175.842,8.330,148.434
C04988=1206.845,400.401,-81.245,-175.842,8.327,148.433
C04989=1206.848,400.153,-81.209,-175.843,8.324,148.432
C04990=1206.852,399.906,-81.176,-175.844,8.322,148.432
C04991=1206.856,399.658,-81.141,-175.844,8.320,148.432
C04992=1206.860,399.411,-81.106,-175.845,8.317,148.431
C04993=1206.864,399.163,-81.071,-175.845,8.315,148.430
C04994=1206.869,398.916,-81.036,-175.845,8.313,148.430
C04995=1206.873,398.668,-81.001,-175.846,8.309,148.429
C04996=1206.876,398.421,-80.967,-175.846,8.307,148.429
C04997=1206.880,398.173,-80.932,-175.847,8.305,148.428
C04998=1206.885,397.925,-80.897,-175.848,8.302,148.428
C04999=1206.889,397.678,-80.862,-175.848,8.300,148.427
C05000=1206.893,397.430,-80.827,-175.849,8.297,148.427
C05001=1206.896,397.183,-80.793,-175.849,8.294,148.426
C05002=1206.901,396.935,-80.759,-175.850,8.293,148.426
C05003=1206.905,396.688,-80.723,-175.850,8.289,148.425
C05004=1206.909,396.440,-80.689,-175.851,8.287,148.425
C05005=1206.913,396.192,-80.654,-175.852,8.284,148.425
C05006=1206.917,395.945,-80.620,-175.852,8.282,148.424
C05007=1206.921,395.698,-80.585,-175.852,8.280,148.423
C05008=1206.925,395.450,-80.550,-175.853,8.277,148.423
C05009=1206.929,395.202,-80.515,-175.854,8.275,148.423
C05010=1206.933,394.955,-80.481,-175.854,8.272,148.422
C05011=1206.937,394.707,-80.447,-175.855,8.269,148.421
C05012=1206.941,394.460,-80.411,-175.856,8.267,148.421
C05013=1206.945,394.212,-80.376,-175.856,8.264,148.420
C05014=1206.949,393.965,-80.343,-175.857,8.261,148.420
C05015=1206.953,393.717,-80.308,-175.857,8.259,148.419
C05016=1206.958,393.469,-80.273,-175.858,8.256,148.419
C05017=1206.960,393.222,-80.238,-175.858,8.254,148.418
C05018=1206.966,392.939,-80.199,-175.859,8.251,148.418
C05019=1206.971,392.657,-80.159,-175.860,8.248,148.417
C05020=1206.975,392.374,-80.120,-175.861,8.244,148.417
C05021=1206.980,392.092,-80.080,-175.862,8.241,148.416
C05022=1206.983,391.845,-80.046,-175.862,8.239,148.416
C05023=1206.987,391.597,-80.012,-175.863,8.236,148.415
C05024=1206.992,391.349,-79.977,-175.864,8.233,148.414
C05025=1206.995,391.101,-79.943,-175.864,8.231,148.414
C05026=1207.000,390.854,-79.908,-175.865,8.228,148.414
C05027=1207.004,390.607,-79.874,-175.865,8.226,148.413
C05028=1207.008,390.359,-79.840,-175.867,8.223,148.413
C05029=1207.012,390.111,-79.805,-175.867,8.220,148.412
C05030=1207.016,389.864,-79.770,-175.868,8.218,148.412
C05031=1207.020,389.617,-79.736,-175.869,8.215,148.411
C05032=1207.024,389.369,-79.701,-175.869,8.212,148.411
C05033=1207.028,389.121,-79.667,-175.870,8.210,148.410
C05034=1207.031,388.873,-79.632,-175.871,8.207,148.410
C05035=1207.036,388.626,-79.598,-175.872,8.204,148.409
C05036=1207.040,388.378,-79.563,-175.872,8.202,148.409
C05037=1207.044,388.131,-79.529,-175.873,8.198,148.408
C05038=1207.048,387.883,-79.495,-175.874,8.196,148.408
C05039=1207.052,387.635,-79.460,-175.875,8.193,148.407
C05040=1207.056,387.388,-79.426,-175.876,8.191,148.407
C05041=1207.061,387.141,-79.391,-175.876,8.187,148.406
C05042=1207.064,386.893,-79.357,-175.877,8.184,148.406
C05043=1207.068,386.645,-79.323,-175.878,8.182,148.405
C05044=1207.072,386.397,-79.288,-175.879,8.179,148.405
C05045=1207.076,386.150,-79.254,-175.880,8.176,148.404
C05046=1207.081,385.903,-79.220,-175.881,8.173,148.404
C05047=1207.084,385.654,-79.186,-175.881,8.171,148.403
C05048=1207.089,385.407,-79.152,-175.882,8.168,148.403
C05049=1207.093,385.159,-79.117,-175.883,8.165,148.402
C05050=1207.097,384.912,-79.083,-175.884,8.162,148.402
C05051=1207.101,384.664,-79.048,-175.885,8.160,148.401
C05052=1207.105,384.416,-79.014,-175.885,8.157,148.401
C05053=1207.109,384.169,-78.980,-175.887,8.154,148.400
C05054=1207.113,383.922,-78.946,-175.887,8.151,148.400
C05055=1207.117,383.674,-78.911,-175.889,8.149,148.399
C05056=1207.121,383.427,-78.877,-175.889,8.145,148.399
C05057=1207.126,383.179,-78.843,-175.891,8.143,148.398
C05058=1207.129,382.931,-78.809,-175.892,8.140,148.398
C05059=1207.133,382.683,-78.775,-175.893,8.137,148.397
C05060=1207.137,382.435,-78.740,-175.893,8.135,148.397
C05061=1207.141,382.188,-78.706,-175.894,8.132,148.397
C05062=1207.146,381.941,-78.672,-175.895,8.129,148.396
C05063=1207.149,381.692,-78.638,-175.896,8.126,148.396
C05064=1207.154,381.445,-78.604,-175.897,8.123,148.395
C05065=1207.158,381.198,-78.570,-175.898,8.120,148.395
C05066=1207.162,380.950,-78.535,-175.899,8.117,148.394
C05067=1207.166,380.702,-78.502,-175.900,8.114,148.394
C05068=1207.170,380.455,-78.467,-175.902,8.111,148.393
C05069=1207.174,380.207,-78.433,-175.902,8.108,148.393
C05070=1207.178,379.959,-78.399,-175.903,8.105,148.392
C05071=1207.182,379.712,-78.365,-175.905,8.103,148.392
C05072=1207.186,379.464,-78.332,-175.905,8.100,148.391
C05073=1207.190,379.216,-78.297,-175.907,8.097,148.391
C05074=1207.194,378.969,-78.263,-175.908,8.094,148.391
C05075=1207.199,378.721,-78.229,-175.909,8.091,148.390
C05076=1207.202,378.473,-78.195,-175.910,8.088,148.390
C05077=1207.207,378.226,-78.160,-175.911,8.085,148.389
C05078=1207.211,377.978,-78.127,-175.912,8.082,148.389
C05079=1207.214,377.730,-78.093,-175.913,8.079,148.388
C05080=1207.219,377.483,-78.058,-175.914,8.076,148.388
C05081=1207.223,377.235,-78.025,-175.915,8.074,148.387
C05082=1207.227,376.988,-77.991,-175.917,8.071,148.387
C05083=1207.231,376.740,-77.957,-175.917,8.068,148.386
C05084=1207.235,376.492,-77.923,-175.919,8.065,148.386
C05085=1207.239,376.245,-77.889,-175.920,8.062,148.386
C05086=1207.243,375.998,-77.855,-175.922,8.059,148.385
C05087=1207.247,375.749,-77.821,-175.923,8.056,148.385
C05088=1207.251,375.502,-77.787,-175.924,8.053,148.384
C05089=1207.255,375.254,-77.754,-175.925,8.050,148.384
C05090=1207.259,375.006,-77.719,-175.926,8.047,148.384
C05091=1207.263,374.758,-77.686,-175.927,8.044,148.383
C05092=1207.267,374.511,-77.652,-175.928,8.041,148.383
C05093=1207.272,374.264,-77.618,-175.930,8.039,148.382
C05094=1207.276,374.016,-77.585,-175.931,8.035,148.382
C05095=1207.279,373.768,-77.550,-175.933,8.032,148.381
C05096=1207.284,373.520,-77.517,-175.934,8.029,148.381
C05097=1207.288,373.273,-77.483,-175.935,8.026,148.381
C05098=1207.292,373.025,-77.449,-175.936,8.024,148.380
C05099=1207.296,372.777,-77.415,-175.938,8.020,148.380
C05100=1207.300,372.530,-77.382,-175.939,8.017,148.379
C05101=1207.304,372.282,-77.348,-175.940,8.014,148.379
C05102=1207.309,372.034,-77.314,-175.941,8.011,148.379
C05103=1207.313,371.787,-77.281,-175.942,8.008,148.378
C05104=1207.316,371.539,-77.246,-175.944,8.005,148.378
C05105=1207.320,371.291,-77.213,-175.946,8.002,148.377
C05106=1207.325,371.044,-77.179,-175.947,8.000,148.377
C05107=1207.329,370.796,-77.146,-175.948,7.997,148.377
C05108=1207.333,370.549,-77.112,-175.950,7.993,148.376
C05109=1207.336,370.300,-77.078,-175.951,7.990,148.376
C05110=1207.341,370.052,-77.045,-175.952,7.987,148.375
C05111=1207.345,369.805,-77.011,-175.953,7.985,148.375
C05112=1207.349,369.558,-76.978,-175.955,7.981,148.375
C05113=1207.353,369.310,-76.944,-175.956,7.978,148.374
C05114=1207.357,369.062,-76.910,-175.958,7.975,148.374
C05115=1207.362,368.814,-76.876,-175.959,7.972,148.373
C05116=1207.366,368.566,-76.843,-175.961,7.969,148.373
C05117=1207.369,368.319,-76.809,-175.962,7.966,148.373
C05118=1207.374,368.071,-76.776,-175.964,7.963,148.372
C05119=1207.378,367.824,-76.743,-175.965,7.960,148.372
C05120=1207.382,367.576,-76.709,-175.966,7.957,148.372
C05121=1207.386,367.328,-76.675,-175.968,7.953,148.371
C05122=1207.390,367.048,-76.638,-175.969,7.951,148.371
C05123=1207.396,366.767,-76.600,-175.972,7.947,148.371
C05124=1207.400,366.487,-76.562,-175.973,7.944,148.370
C05125=1207.405,366.207,-76.524,-175.975,7.940,148.370
C05126=1207.408,365.958,-76.490,-175.976,7.937,148.369
C05127=1207.413,365.711,-76.457,-175.978,7.934,148.369
C05128=1207.417,365.463,-76.424,-175.980,7.931,148.369
C05129=1207.421,365.216,-76.390,-175.981,7.928,148.368
C05130=1207.425,364.968,-76.357,-175.983,7.925,148.368
C05131=1207.429,364.720,-76.324,-175.984,7.922,148.368
C05132=1207.433,364.473,-76.291,-175.986,7.919,148.367
C05133=1207.437,364.225,-76.257,-175.987,7.916,148.367
C05134=1207.442,363.977,-76.224,-175.989,7.913,148.367
C05135=1207.445,363.729,-76.189,-175.991,7.909,148.366
C05136=1207.449,363.481,-76.156,-175.992,7.907,148.366
C05137=1207.453,363.234,-76.123,-175.994,7.903,148.366
C05138=1207.458,362.986,-76.090,-175.995,7.900,148.365
C05139=1207.462,362.738,-76.057,-175.997,7.898,148.365
C05140=1207.466,362.490,-76.024,-175.999,7.894,148.365
C05141=1207.470,362.243,-75.990,-176.000,7.892,148.364
C05142=1207.474,361.995,-75.957,-176.002,7.888,148.364
C05143=1207.478,361.747,-75.924,-176.003,7.885,148.364
C05144=1207.482,361.499,-75.891,-176.006,7.882,148.363
C05145=1207.487,361.252,-75.858,-176.007,7.879,148.363
C05146=1207.491,361.004,-75.825,-176.009,7.876,148.363
C05147=1207.495,360.756,-75.792,-176.010,7.873,148.362
C05148=1207.499,360.509,-75.758,-176.011,7.870,148.362
C05149=1207.503,360.261,-75.725,-176.014,7.867,148.362
C05150=1207.507,360.013,-75.692,-176.015,7.864,148.361
C05151=1207.511,359.765,-75.659,-176.017,7.861,148.361
C05152=1207.516,359.518,-75.626,-176.019,7.858,148.361
C05153=1207.520,359.270,-75.593,-176.020,7.855,148.360
C05154=1207.523,359.021,-75.559,-176.022,7.852,148.360
C05155=1207.527,358.774,-75.526,-176.024,7.848,148.360
C05156=1207.531,358.526,-75.493,-176.026,7.846,148.360
C05157=1207.535,358.279,-75.460,-176.027,7.842,148.359
C05158=1207.539,358.030,-75.428,-176.029,7.840,148.359
C05159=1207.543,357.783,-75.395,-176.031,7.836,148.359
C05160=1207.548,357.535,-75.361,-176.032,7.834,148.358
C05161=1207.552,357.288,-75.329,-176.035,7.830,148.358
C05162=1207.556,357.040,-75.296,-176.036,7.828,148.358
C05163=1207.561,356.792,-75.262,-176.038,7.824,148.358
C05164=1207.565,356.544,-75.230,-176.040,7.822,148.357
C05165=1207.569,356.296,-75.197,-176.041,7.818,148.357
C05166=1207.573,356.049,-75.164,-176.044,7.815,148.357
C05167=1207.577,355.801,-75.131,-176.045,7.812,148.357
C05168=1207.581,355.553,-75.098,-176.047,7.809,148.356
C05169=1207.585,355.305,-75.065,-176.049,7.806,148.356
C05170=1207.589,355.057,-75.032,-176.051,7.803,148.356
C05171=1207.594,354.810,-74.999,-176.053,7.800,148.355
C05172=1207.597,354.562,-74.967,-176.054,7.796,148.355
C05173=1207.601,354.314,-74.934,-176.056,7.794,148.355
C05174=1207.606,354.066,-74.901,-176.058,7.791,148.355
C05175=1207.610,353.818,-74.868,-176.060,7.788,148.354
C05176=1207.614,353.570,-74.835,-176.062,7.784,148.354
C05177=1207.618,353.323,-74.803,-176.063,7.782,148.354
C05178=1207.622,353.075,-74.770,-176.065,7.779,148.354
C05179=1207.627,352.827,-74.738,-176.067,7.776,148.353
C05180=1207.631,352.579,-74.704,-176.069,7.773,148.353
C05181=1207.634,352.332,-74.672,-176.071,7.769,148.353
C05182=1207.639,352.084,-74.639,-176.073,7.767,148.353
C05183=1207.643,351.836,-74.606,-176.075,7.763,148.352
C05184=1207.647,351.588,-74.574,-176.077,7.761,148.352
C05185=1207.651,351.340,-74.541,-176.079,7.757,148.352
C05186=1207.655,351.092,-74.509,-176.080,7.755,148.352
C05187=1207.659,350.844,-74.476,-176.082,7.751,148.351
C05188=1207.664,350.597,-74.443,-176.084,7.749,148.351
C05189=1207.668,350.349,-74.411,-176.086,7.745,148.351
C05190=1207.672,350.101,-74.378,-176.088,7.743,148.351
C05191=1207.676,349.853,-74.345,-176.090,7.739,148.351
C05192=1207.680,349.606,-74.313,-176.092,7.736,148.350
C05193=1207.684,349.357,-74.280,-176.094,7.734,148.350
C05194=1207.688,349.109,-74.247,-176.096,7.730,148.350
C05195=1207.693,348.862,-74.216,-176.098,7.728,148.350
C05196=1207.697,348.614,-74.183,-176.099,7.724,148.349
C05197=1207.701,348.366,-74.150,-176.101,7.722,148.349
C05198=1207.705,348.118,-74.118,-176.103,7.718,148.349
C05199=1207.709,347.870,-74.085,-176.105,7.716,148.349
C05200=1207.713,347.622,-74.053,-176.107,7.712,148.348
C05201=1207.718,347.375,-74.021,-176.109,7.709,148.348
C05202=1207.722,347.127,-73.988,-176.111,7.707,148.348
C05203=1207.726,346.879,-73.956,-176.113,7.703,148.348
C05204=1207.730,346.631,-73.923,-176.115,7.701,148.348
C05205=1207.734,346.383,-73.891,-176.117,7.697,148.347
C05206=1207.739,346.135,-73.859,-176.119,7.695,148.347
C05207=1207.743,345.888,-73.826,-176.121,7.691,148.347
C05208=1207.746,345.640,-73.794,-176.123,7.688,148.347
C05209=1207.751,345.391,-73.762,-176.125,7.686,148.347
C05210=1207.755,345.144,-73.730,-176.127,7.682,148.346
C05211=1207.759,344.896,-73.697,-176.129,7.680,148.346
C05212=1207.764,344.648,-73.665,-176.131,7.676,148.346
C05213=1207.767,344.400,-73.633,-176.133,7.674,148.346
C05214=1207.772,344.153,-73.600,-176.135,7.671,148.346
C05215=1207.776,343.905,-73.568,-176.137,7.668,148.346
C05216=1207.780,343.656,-73.536,-176.139,7.665,148.345
C05217=1207.784,343.408,-73.504,-176.141,7.662,148.345
C05218=1207.789,343.161,-73.472,-176.143,7.659,148.345
C05219=1207.792,342.913,-73.439,-176.145,7.656,148.345
C05220=1207.797,342.665,-73.407,-176.147,7.652,148.345
C05221=1207.801,342.417,-73.375,-176.149,7.650,148.344
C05222=1207.806,342.169,-73.343,-176.151,7.647,148.344
C05223=1207.809,341.921,-73.311,-176.153,7.644,148.344
C05224=1207.814,341.673,-73.279,-176.156,7.641,148.344
C05225=1207.818,341.426,-73.247,-176.157,7.639,148.344
C05226=1207.823,341.147,-73.211,-176.160,7.634,148.344
C05227=1207.827,340.869,-73.175,-176.162,7.631,148.343
C05228=1207.832,340.592,-73.139,-176.164,7.628,148.343
C05229=1207.837,340.312,-73.103,-176.167,7.625,148.343
C05230=1207.840,340.064,-73.071,-176.169,7.622,148.343
C05231=1207.845,339.817,-73.040,-176.171,7.619,148.343
C05232=1207.849,339.569,-73.007,-176.173,7.616,148.342
C05233=1207.853,339.321,-72.975,-176.175,7.613,148.342
C05234=1207.858,339.073,-72.943,-176.178,7.610,148.342
C05235=1207.862,338.825,-72.911,-176.179,7.607,148.342
C05236=1207.865,338.577,-72.880,-176.181,7.604,148.342
C05237=1207.870,338.329,-72.848,-176.183,7.602,148.342
C05238=1207.874,338.081,-72.816,-176.186,7.598,148.342
C05239=1207.878,337.833,-72.784,-176.187,7.596,148.342
C05240=1207.883,337.586,-72.752,-176.190,7.593,148.341
C05241=1207.887,337.338,-72.720,-176.192,7.589,148.341
C05242=1207.891,337.090,-72.688,-176.194,7.587,148.341
C05243=1207.895,336.842,-72.656,-176.196,7.584,148.341
C05244=1207.899,336.594,-72.624,-176.198,7.581,148.341
C05245=1207.903,336.346,-72.593,-176.200,7.578,148.341
C05246=1207.907,336.098,-72.561,-176.203,7.575,148.340
C05247=1207.912,335.849,-72.529,-176.204,7.572,148.340
C05248=1207.916,335.602,-72.498,-176.207,7.569,148.340
C05249=1207.920,335.354,-72.466,-176.209,7.567,148.340
C05250=1207.924,335.107,-72.434,-176.211,7.563,148.340
C05251=1207.928,334.858,-72.402,-176.214,7.560,148.340
C05252=1207.932,334.610,-72.370,-176.215,7.558,148.340
C05253=1207.937,334.362,-72.339,-176.217,7.555,148.340
C05254=1207.941,334.114,-72.307,-176.220,7.552,148.340
C05255=1207.946,333.867,-72.275,-176.222,7.549,148.339
C05256=1207.949,333.619,-72.243,-176.224,7.546,148.339
C05257=1207.954,333.371,-72.213,-176.226,7.543,148.339
C05258=1207.958,333.123,-72.181,-176.228,7.540,148.339
C05259=1207.961,332.875,-72.149,-176.230,7.538,148.339
C05260=1207.966,332.627,-72.118,-176.233,7.535,148.339
C05261=1207.970,332.378,-72.086,-176.235,7.531,148.339
C05262=1207.975,332.131,-72.054,-176.237,7.529,148.339
C05263=1207.979,331.882,-72.023,-176.239,7.526,148.338
C05264=1207.983,331.635,-71.992,-176.241,7.523,148.338
C05265=1207.987,331.387,-71.960,-176.243,7.520,148.338
C05266=1207.991,331.139,-71.929,-176.246,7.517,148.338
C05267=1207.995,330.891,-71.897,-176.248,7.515,148.338
C05268=1208.000,330.643,-71.865,-176.250,7.511,148.338
C05269=1208.004,330.395,-71.834,-176.252,7.509,148.338
C05270=1208.008,330.147,-71.803,-176.254,7.506,148.338
C05271=1208.012,329.899,-71.771,-176.257,7.503,148.338
C05272=1208.017,329.651,-71.740,-176.259,7.500,148.337
C05273=1208.021,329.403,-71.709,-176.261,7.497,148.337
C05274=1208.025,329.155,-71.677,-176.263,7.495,148.337
C05275=1208.029,328.907,-71.646,-176.265,7.491,148.337
C05276=1208.033,328.659,-71.615,-176.268,7.488,148.337
C05277=1208.037,328.411,-71.583,-176.270,7.486,148.337
C05278=1208.042,328.163,-71.552,-176.272,7.483,148.337
C05279=1208.046,327.915,-71.521,-176.274,7.480,148.337
C05280=1208.050,327.667,-71.490,-176.277,7.477,148.337
C05281=1208.054,327.419,-71.458,-176.279,7.474,148.337
C05282=1208.058,327.171,-71.427,-176.281,7.472,148.337
C05283=1208.062,326.923,-71.396,-176.284,7.468,148.337
C05284=1208.067,326.675,-71.364,-176.285,7.466,148.336
C05285=1208.071,326.427,-71.334,-176.288,7.463,148.336
C05286=1208.075,326.179,-71.302,-176.290,7.460,148.336
C05287=1208.080,325.931,-71.271,-176.292,7.457,148.336
C05288=1208.084,325.683,-71.240,-176.294,7.454,148.336
C05289=1208.088,325.435,-71.208,-176.297,7.452,148.336
C05290=1208.092,325.187,-71.177,-176.299,7.448,148.336
C05291=1208.096,324.939,-71.146,-176.301,7.445,148.336
C05292=1208.101,324.691,-71.115,-176.304,7.443,148.336
C05293=1208.105,324.443,-71.084,-176.306,7.440,148.336
C05294=1208.109,324.195,-71.053,-176.308,7.438,148.336
C05295=1208.113,323.946,-71.022,-176.310,7.434,148.335
C05296=1208.117,323.699,-70.991,-176.313,7.431,148.335
C05297=1208.122,323.451,-70.960,-176.315,7.429,148.336
C05298=1208.126,323.203,-70.929,-176.317,7.426,148.335
C05299=1208.130,322.955,-70.898,-176.319,7.424,148.335
C05300=1208.134,322.707,-70.867,-176.321,7.420,148.335
C05301=1208.139,322.459,-70.836,-176.324,7.417,148.335
C05302=1208.143,322.211,-70.805,-176.326,7.415,148.335
C05303=1208.146,321.962,-70.774,-176.328,7.412,148.335
C05304=1208.151,321.714,-70.744,-176.331,7.409,148.335
C05305=1208.155,321.467,-70.712,-176.333,7.406,148.335
C05306=1208.159,321.218,-70.681,-176.335,7.403,148.335
C05307=1208.164,320.970,-70.650,-176.338,7.401,148.335
C05308=1208.169,320.722,-70.620,-176.340,7.398,148.335
C05309=1208.172,320.474,-70.589,-176.342,7.395,148.335
C05310=1208.177,320.226,-70.558,-176.345,7.392,148.335
C05311=1208.181,319.978,-70.528,-176.347,7.389,148.335
C05312=1208.185,319.729,-70.496,-176.349,7.387,148.335
C05313=1208.189,319.482,-70.466,-176.352,7.384,148.335
C05314=1208.194,319.234,-70.435,-176.354,7.381,148.335
C05315=1208.197,318.986,-70.404,-176.356,7.378,148.334
C05316=1208.202,318.738,-70.373,-176.359,7.375,148.334
C05317=1208.206,318.490,-70.343,-176.361,7.373,148.334
C05318=1208.210,318.242,-70.312,-176.363,7.370,148.334
C05319=1208.214,317.994,-70.281,-176.365,7.367,148.334
C05320=1208.219,317.746,-70.250,-176.368,7.364,148.334
C05321=1208.223,317.498,-70.220,-176.370,7.361,148.334
C05322=1208.227,317.249,-70.189,-176.373,7.359,148.334
C05323=1208.232,317.001,-70.159,-176.375,7.356,148.334
C05324=1208.236,316.753,-70.129,-176.377,7.354,148.334
C05325=1208.240,316.505,-70.098,-176.380,7.351,148.334
C05326=1208.244,316.256,-70.067,-176.382,7.347,148.334
C05327=1208.248,316.009,-70.036,-176.384,7.345,148.334
C05328=1208.253,315.761,-70.006,-176.387,7.342,148.334
C05329=1208.257,315.513,-69.975,-176.389,7.340,148.334
C05330=1208.262,315.237,-69.942,-176.391,7.337,148.334
C05331=1208.266,314.960,-69.907,-176.394,7.334,148.334
C05332=1208.271,314.685,-69.873,-176.396,7.330,148.334
C05333=1208.276,314.408,-69.839,-176.399,7.327,148.334
C05334=1208.280,314.160,-69.809,-176.402,7.324,148.334
C05335=1208.284,313.913,-69.779,-176.404,7.322,148.334
C05336=1208.289,313.665,-69.748,-176.406,7.319,148.334
C05337=1208.293,313.416,-69.718,-176.409,7.316,148.334
C05338=1208.297,313.168,-69.687,-176.411,7.313,148.334
C05339=1208.302,312.920,-69.656,-176.413,7.310,148.334
C05340=1208.306,312.671,-69.627,-176.416,7.308,148.334
C05341=1208.311,312.423,-69.596,-176.418,7.305,148.334
C05342=1208.314,312.175,-69.566,-176.420,7.303,148.334
C05343=1208.318,311.927,-69.535,-176.423,7.300,148.334
C05344=1208.323,311.679,-69.505,-176.425,7.297,148.334
C05345=1208.327,311.431,-69.475,-176.427,7.294,148.334
C05346=1208.331,311.183,-69.445,-176.430,7.291,148.334
C05347=1208.336,310.935,-69.414,-176.432,7.289,148.334
C05348=1208.340,310.687,-69.384,-176.435,7.286,148.334
C05349=1208.344,310.438,-69.353,-176.437,7.284,148.334
C05350=1208.348,310.190,-69.324,-176.440,7.281,148.334
C05351=1208.353,309.942,-69.293,-176.442,7.278,148.334
C05352=1208.357,309.694,-69.264,-176.444,7.275,148.334
C05353=1208.362,309.446,-69.233,-176.447,7.272,148.334
C05354=1208.366,309.198,-69.203,-176.449,7.270,148.334
C05355=1208.370,308.950,-69.173,-176.452,7.267,148.334
C05356=1208.374,308.702,-69.142,-176.454,7.265,148.334
C05357=1208.378,308.453,-69.113,-176.456,7.262,148.334
C05358=1208.382,308.205,-69.082,-176.459,7.259,148.334
C05359=1208.387,307.957,-69.052,-176.461,7.257,148.334
C05360=1208.391,307.709,-69.022,-176.464,7.254,148.334
C05361=1208.395,307.461,-68.992,-176.465,7.251,148.334
C05362=1208.400,307.212,-68.963,-176.468,7.248,148.334
C05363=1208.404,306.964,-68.932,-176.470,7.246,148.334
C05364=1208.408,306.716,-68.902,-176.473,7.243,148.334
C05365=1208.412,306.469,-68.872,-176.476,7.240,148.334
C05366=1208.417,306.220,-68.842,-176.478,7.238,148.334
C05367=1208.421,305.972,-68.812,-176.480,7.235,148.334
C05368=1208.426,305.724,-68.782,-176.483,7.232,148.334
C05369=1208.430,305.475,-68.753,-176.485,7.229,148.334
C05370=1208.434,305.228,-68.722,-176.487,7.227,148.334
C05371=1208.438,304.980,-68.693,-176.490,7.224,148.334
C05372=1208.443,304.731,-68.663,-176.492,7.222,148.334
C05373=1208.447,304.483,-68.633,-176.495,7.219,148.334
C05374=1208.451,304.235,-68.603,-176.497,7.217,148.334
C05375=1208.456,303.986,-68.573,-176.500,7.214,148.334
C05376=1208.460,303.739,-68.543,-176.502,7.211,148.334
C05377=1208.464,303.491,-68.514,-176.504,7.208,148.334
C05378=1208.468,303.242,-68.484,-176.507,7.205,148.334
C05379=1208.473,302.994,-68.454,-176.509,7.203,148.334
C05380=1208.477,302.746,-68.424,-176.512,7.200,148.334
C05381=1208.481,302.498,-68.394,-176.514,7.198,148.334
C05382=1208.485,302.250,-68.365,-176.517,7.195,148.334
C05383=1208.490,302.001,-68.335,-176.519,7.193,148.334
C05384=1208.494,301.753,-68.305,-176.522,7.190,148.334
C05385=1208.498,301.505,-68.275,-176.524,7.188,148.335
C05386=1208.503,301.257,-68.246,-176.526,7.184,148.335
C05387=1208.507,301.008,-68.216,-176.529,7.181,148.335
C05388=1208.512,300.760,-68.186,-176.531,7.179,148.335
C05389=1208.516,300.512,-68.157,-176.534,7.176,148.335
C05390=1208.520,300.263,-68.127,-176.536,7.174,148.335
C05391=1208.524,300.016,-68.097,-176.539,7.171,148.335
C05392=1208.528,299.767,-68.068,-176.541,7.169,148.335
C05393=1208.532,299.519,-68.038,-176.544,7.166,148.335
C05394=1208.537,299.271,-68.008,-176.546,7.164,148.335
C05395=1208.541,299.022,-67.979,-176.548,7.161,148.335
C05396=1208.546,298.774,-67.949,-176.550,7.158,148.335
C05397=1208.550,298.526,-67.920,-176.553,7.155,148.335
C05398=1208.554,298.278,-67.891,-176.555,7.153,148.335
C05399=1208.559,298.030,-67.861,-176.558,7.150,148.335
C05400=1208.563,297.782,-67.832,-176.560,7.148,148.335
C05401=1208.567,297.533,-67.803,-176.563,7.145,148.335
C05402=1208.571,297.285,-67.773,-176.565,7.143,148.335
C05403=1208.575,297.037,-67.744,-176.568,7.140,148.335
C05404=1208.580,296.789,-67.714,-176.570,7.138,148.335
C05405=1208.584,296.540,-67.685,-176.573,7.135,148.335
C05406=1208.588,296.292,-67.655,-176.576,7.132,148.335
C05407=1208.592,296.044,-67.626,-176.578,7.130,148.336
C05408=1208.597,295.796,-67.597,-176.580,7.126,148.336
C05409=1208.601,295.548,-67.567,-176.583,7.124,148.336
C05410=1208.606,295.299,-67.539,-176.585,7.121,148.336
C05411=1208.610,295.051,-67.509,-176.587,7.119,148.336
C05412=1208.614,294.803,-67.480,-176.590,7.116,148.336
C05413=1208.618,294.554,-67.450,-176.593,7.114,148.336
C05414=1208.622,294.306,-67.421,-176.595,7.111,148.336
C05415=1208.627,294.058,-67.392,-176.597,7.109,148.336
C05416=1208.632,293.810,-67.363,-176.600,7.106,148.336
C05417=1208.636,293.561,-67.333,-176.602,7.104,148.336
C05418=1208.640,293.313,-67.304,-176.605,7.101,148.336
C05419=1208.644,293.065,-67.275,-176.607,7.098,148.336
C05420=1208.649,292.817,-67.245,-176.610,7.095,148.336
C05421=1208.653,292.568,-67.217,-176.612,7.094,148.337
C05422=1208.658,292.320,-67.187,-176.615,7.091,148.337
C05423=1208.662,292.072,-67.158,-176.617,7.088,148.337
C05424=1208.666,291.823,-67.129,-176.620,7.085,148.337
C05425=1208.671,291.575,-67.100,-176.622,7.083,148.337
C05426=1208.675,291.327,-67.071,-176.625,7.080,148.337
C05427=1208.679,291.079,-67.042,-176.627,7.078,148.337
C05428=1208.683,290.830,-67.013,-176.630,7.075,148.337
C05429=1208.687,290.582,-66.983,-176.632,7.073,148.337
C05430=1208.692,290.334,-66.954,-176.634,7.071,148.337
C05431=1208.697,290.086,-66.926,-176.637,7.068,148.337
C05432=1208.701,289.837,-66.896,-176.639,7.066,148.337
C05433=1208.705,289.589,-66.868,-176.642,7.063,148.338
C05434=1208.710,289.315,-66.835,-176.645,7.060,148.338
C05435=1208.715,289.040,-66.803,-176.648,7.057,148.338
C05436=1208.719,288.766,-66.772,-176.650,7.055,148.338
C05437=1208.724,288.492,-66.739,-176.653,7.052,148.338
C05438=1208.729,288.244,-66.711,-176.656,7.049,148.338
C05439=1208.732,287.996,-66.682,-176.658,7.047,148.338
C05440=1208.737,287.747,-66.654,-176.660,7.044,148.338
C05441=1208.741,287.499,-66.624,-176.663,7.042,148.338
C05442=1208.746,287.251,-66.596,-176.666,7.039,148.338
C05443=1208.750,287.002,-66.566,-176.668,7.037,148.338
C05444=1208.754,286.754,-66.538,-176.670,7.034,148.338
C05445=1208.759,286.506,-66.510,-176.673,7.032,148.339
C05446=1208.763,286.257,-66.480,-176.675,7.029,148.339
C05447=1208.767,286.009,-66.452,-176.678,7.026,148.339
C05448=1208.772,285.761,-66.423,-176.680,7.024,148.339
C05449=1208.776,285.512,-66.394,-176.683,7.021,148.339
C05450=1208.781,285.264,-66.365,-176.685,7.019,148.339
C05451=1208.785,285.016,-66.337,-176.688,7.016,148.339
C05452=1208.789,284.767,-66.308,-176.690,7.014,148.339
C05453=1208.794,284.519,-66.279,-176.693,7.011,148.339
C05454=1208.798,284.271,-66.251,-176.695,7.009,148.340
C05455=1208.802,284.022,-66.222,-176.698,7.006,148.340
C05456=1208.806,283.774,-66.193,-176.700,7.004,148.340
C05457=1208.811,283.526,-66.165,-176.702,7.002,148.340
C05458=1208.815,283.277,-66.136,-176.706,6.999,148.340
C05459=1208.820,283.030,-66.108,-176.708,6.997,148.340
C05460=1208.824,282.781,-66.079,-176.710,6.994,148.340
C05461=1208.829,282.532,-66.050,-176.712,6.992,148.340
C05462=1208.833,282.284,-66.023,-176.716,6.989,148.340
C05463=1208.837,282.036,-65.993,-176.718,6.987,148.340
C05464=1208.841,281.788,-65.965,-176.720,6.984,148.340
C05465=1208.846,281.539,-65.937,-176.723,6.982,148.341
C05466=1208.850,281.290,-65.908,-176.725,6.980,148.341
C05467=1208.855,281.043,-65.880,-176.728,6.977,148.341
C05468=1208.859,280.794,-65.851,-176.730,6.974,148.341
C05469=1208.863,280.546,-65.823,-176.733,6.972,148.341
C05470=1208.868,280.298,-65.794,-176.735,6.970,148.341
C05471=1208.871,280.049,-65.766,-176.738,6.967,148.341
